Yaskawa INFORM job: ARIEL_TEST.JBI

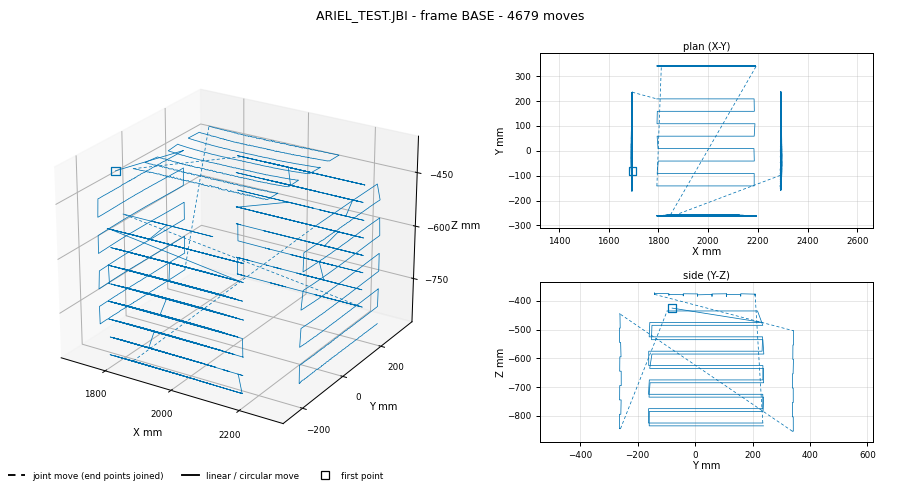
[picture p0: tool path of ARIEL_TEST.JBI in frame BASE, 4679 of 4679 moves have a stored position in this frame; points joined in program order, loops and branches not executed]
/JOB
//NAME ARIEL_TEST
//POS
///NPOS 4679,0,0,0,0,0
///TOOL 0
///POSTYPE BASE
///RECTAN
///RCONF 1,0,0,0,0,0,0,0,0,0,0,0,0,0,0,0,0,0,0,0,0,0,0,0
C00000=1696.132,-80.047,-425.128,-2.7960,72.8573,-92.9280
C00001=1694.988,235.674,-475.128,91.6331,81.5548,1.6157
C00002=1694.763,232.398,-475.128,113.1075,87.8917,23.0901
C00003=1694.793,228.055,-475.128,-70.6571,88.5964,-160.6630
C00004=1695.151,224.781,-475.128,-66.4401,88.6995,-156.4461
C00005=1695.130,221.009,-475.128,-43.9344,88.9803,-133.9346
C00006=1695.054,219.997,-475.128,-8.9266,88.7912,-98.9268
C00007=1695.058,217.094,-475.128,-159.0817,88.5678,110.9246
C00008=1694.887,215.803,-475.128,-11.6768,88.8428,-101.6770
C00009=1695.188,212.462,-475.128,-4.3716,86.4536,-94.3776
C00010=1695.133,208.131,-475.128,-42.6337,89.3986,-132.6340
C00011=1695.189,206.048,-475.128,-13.4931,89.5876,-103.4933
C00012=1695.116,201.470,-475.128,50.1911,88.5907,-39.8033
C00013=1694.965,197.460,-475.128,48.4607,89.2725,-41.5394
C00014=1695.140,191.185,-475.128,17.4924,89.6392,-72.5020
C00015=1694.918,187.331,-475.128,31.8851,88.8600,-58.1093
C00016=1695.110,184.389,-475.128,64.8530,89.3642,-25.1471
C00017=1694.969,179.240,-475.128,-12.1008,87.9146,-102.1068
C00018=1695.056,175.417,-475.128,38.8981,88.5907,-51.0906
C00019=1694.747,170.987,-475.128,47.6299,87.8172,-42.3473
C00020=1694.650,164.775,-475.128,16.4324,88.5105,-73.5620
C00021=1694.533,162.575,-475.128,42.0894,88.3901,-47.8992
C00022=1694.373,158.045,-475.128,56.9978,88.5563,-32.9909
C00023=1695.089,155.989,-475.128,-6.3483,88.3443,-96.3543
C00024=1695.185,152.477,-475.128,-65.8099,88.1495,-155.8216
C00025=1694.724,149.203,-475.128,6.0332,87.2614,-83.9612
C00026=1695.104,146.728,-475.128,19.4862,88.9230,-70.5139
C00027=1694.834,143.853,-475.128,47.7331,88.7053,-42.2556
C00028=1693.934,141.094,-475.128,115.7489,87.4906,25.7258
C00029=1693.799,137.257,-475.128,99.1904,86.6713,9.1730
C00030=1693.895,133.651,-475.128,38.0386,87.8287,-51.9386
C00031=1693.476,130.746,-475.128,21.7208,87.0265,-68.2507
C00032=1694.334,128.603,-475.128,25.3820,86.7859,-64.5838
C00033=1695.164,125.432,-475.128,143.9040,88.7110,53.8981
C00034=1694.863,121.656,-475.128,8.3823,87.0265,-81.6063
C00035=1693.391,117.740,-475.128,20.0649,87.7484,-69.9237
C00036=1694.429,115.474,-475.128,6.2051,87.3817,-83.7893
C00037=1693.264,112.358,-475.128,47.6242,88.3500,-42.3644
C00038=1694.551,109.480,-475.128,-7.0531,87.5078,-97.0590
C00039=1694.104,106.646,-475.128,8.1417,87.1984,-81.8470
C00040=1693.197,102.981,-475.128,-2.9507,87.4448,-92.9509
C00041=1694.004,100.489,-475.128,16.0313,86.9291,-73.9516
C00042=1694.629,96.503,-475.128,0.4354,86.7859,-89.5590
C00043=1693.339,94.279,-475.128,4.1539,86.6025,-85.8405
C00044=1693.243,89.591,-475.128,30.0688,88.3959,-59.9199
C00045=1694.046,86.533,-475.128,-0.4354,87.1010,-90.4356
C00046=1694.079,83.430,-475.128,-14.8969,86.6369,-104.9200
C00047=1694.640,81.259,-475.128,-7.5916,81.0620,-97.6835
C00048=1693.579,77.591,-475.128,-3.7013,86.7286,-93.7072
C00049=1694.579,74.118,-475.128,8.0615,86.6770,-81.9272
C00050=1694.602,71.620,-475.128,5.6550,86.3791,-84.3336
C00051=1693.230,67.936,-475.128,7.5745,86.6827,-82.4085
C00052=1692.692,63.461,-475.128,3.3689,87.3015,-86.6254
C00053=1693.515,60.204,-475.128,-3.5408,86.7515,-93.5410
C00054=1694.397,57.070,-475.128,-1.8678,86.3218,-91.8737
C00055=1695.083,51.313,-475.128,-46.0772,88.8542,-136.0832
C00056=1693.552,49.260,-475.128,3.4492,86.3275,-86.5452
C00057=1693.236,43.220,-475.128,-9.1501,86.3619,-99.1675
C00058=1692.438,40.123,-475.128,-10.2502,86.8604,-100.2676
C00059=1693.005,36.124,-475.128,-0.4583,86.2817,-90.4585
C00060=1694.308,31.082,-475.128,-2.0511,86.4937,-92.0571
C00061=1692.704,27.503,-475.128,2.7845,87.7828,-87.2099
C00062=1693.177,25.817,-475.128,10.8804,87.3073,-79.1082
C00063=1692.952,22.582,-475.128,5.8269,86.0525,-84.1617
C00064=1693.146,20.159,-475.128,3.7700,88.0636,-86.2244
C00065=1694.605,16.625,-475.128,-10.1413,85.7545,-100.1702
C00066=1693.774,12.699,-475.128,-8.9782,86.9578,-98.9899
C00067=1694.221,10.877,-475.128,9.3965,85.4566,-80.5693
C00068=1693.353,8.692,-475.128,-10.5882,87.4791,-100.5999
C00069=1695.395,6.553,-475.128,-14.2781,75.9627,-104.6965
C00070=1694.514,2.859,-475.128,-3.7757,86.2931,-93.7817
C00071=1694.492,-1.569,-475.128,-24.3277,87.2843,-114.3566
C00072=1692.776,-3.735,-475.128,-27.3186,87.2614,-117.3474
C00073=1694.690,-6.961,-475.128,-12.0607,85.7889,-102.0896
C00074=1694.113,-9.973,-475.128,-4.8816,87.4104,-94.8875
C00075=1695.315,-12.616,-475.128,5.5233,88.3386,-84.4711
C00076=1693.186,-16.477,-475.128,-14.8109,86.9692,-104.8283
C00077=1694.776,-17.860,-475.128,-8.1474,86.3963,-98.1591
C00078=1693.169,-22.210,-475.128,-23.4912,87.5364,-113.5086
C00079=1694.236,-24.585,-475.128,-9.7632,86.0238,-99.7863
C00080=1693.849,-28.361,-475.128,-19.7842,87.2041,-109.8073
C00081=1694.081,-32.852,-475.128,-27.7884,87.3932,-117.8173
C00082=1694.169,-36.280,-475.128,-40.8805,87.2156,-130.9151
C00083=1694.436,-38.893,-475.128,-11.4935,86.3332,-101.5166
C00084=1693.377,-42.844,-475.128,-15.4297,87.0208,-105.4528
C00085=1693.729,-46.013,-475.128,-5.6894,87.2843,-95.6954
C00086=1693.512,-48.882,-475.128,-21.3197,87.2729,-111.3371
C00087=1694.121,-53.479,-475.128,-2.0970,87.3703,-92.0972
C00088=1694.254,-55.606,-475.128,-8.6631,87.1239,-98.6747
C00089=1695.480,-60.498,-475.128,-7.5515,88.3615,-97.5517
C00090=1694.880,-63.263,-475.128,-10.0668,86.3447,-100.0899
C00091=1695.519,-67.371,-475.128,-4.2799,86.4650,-94.2916
C00092=1695.154,-69.634,-475.128,-16.6902,86.9062,-106.7133
C00093=1694.837,-73.212,-475.128,-14.3468,87.2099,-104.3642
C00094=1695.406,-77.363,-475.128,-22.5057,86.9921,-112.5346
C00095=1695.106,-81.047,-475.128,-14.6963,88.1438,-104.7023
C00096=1694.416,-84.097,-475.128,-20.3170,87.6281,-110.3344
C00097=1695.519,-87.829,-475.128,82.5403,88.9860,-7.4599
C00098=1694.707,-90.627,-475.128,-9.6600,86.9119,-99.6717
C00099=1695.330,-93.501,-475.128,-21.3369,87.6797,-111.3543
C00100=1695.363,-99.305,-475.128,-13.2009,87.5823,-103.2126
C00101=1694.622,-103.431,-475.128,-32.7502,88.3157,-122.7619
C00102=1695.475,-107.547,-475.128,2.7100,87.8401,-87.2901
C00103=1694.908,-111.406,-475.128,-12.5363,88.2355,-102.5422
C00104=1695.600,-115.157,-475.128,63.4035,89.7939,-26.5967
C00105=1694.895,-121.393,-475.128,-19.4691,88.3730,-109.4750
C00106=1695.267,-125.384,-475.128,-1.8907,88.4245,-91.8967
C00107=1694.736,-129.294,-475.128,-21.9041,89.0491,-111.9101
C00108=1694.843,-133.799,-475.128,-11.6940,88.3558,-101.6942
C00109=1695.271,-139.102,-475.128,-14.4328,88.7511,-104.4387
C00110=1695.095,-144.244,-475.128,-2.4751,88.2813,-92.4753
C00111=1694.850,-148.261,-475.128,-17.9851,88.4532,-107.9910
C00112=1695.327,-150.030,-475.128,46.9596,88.7855,-43.0348
C00113=1695.394,-153.452,-475.128,127.4143,87.1927,37.3854
C00114=1694.805,-157.684,-475.128,-67.2767,86.9635,-157.3055
C00115=1694.500,-159.876,-525.128,-78.9249,82.7121,-169.0110
C00116=1694.421,-156.702,-525.128,-95.0365,88.5391,174.9641
C00117=1694.689,-153.571,-525.128,-16.8220,89.4845,-106.8222
C00118=1694.622,-150.053,-525.128,-18.9878,88.8657,-108.9937
C00119=1694.362,-147.366,-525.128,-40.2216,88.8657,-130.2218
C00120=1694.470,-144.581,-525.128,-53.1189,88.8428,-143.1248
C00121=1694.487,-142.921,-525.128,-69.2419,88.9115,-159.2478
C00122=1694.727,-138.966,-525.128,-58.3614,89.2381,-148.3674
C00123=1694.454,-135.239,-525.128,-40.0268,88.5735,-130.0327
C00124=1694.239,-130.327,-525.128,-74.8282,88.7397,-164.8342
C00125=1694.291,-126.172,-525.128,-35.7353,88.3271,-125.7470
C00126=1693.961,-120.293,-525.128,-44.4557,88.1610,-134.4674
C00127=1694.229,-117.327,-525.128,-39.6773,88.3787,-129.6889
C00128=1693.955,-112.124,-525.128,-39.0126,88.5506,-129.0186
C00129=1694.120,-109.056,-525.128,-37.0875,88.5448,-127.0992
C00130=1693.350,-104.310,-525.128,-49.8072,87.8401,-139.8246
C00131=1693.551,-100.440,-525.128,-37.3396,87.8000,-127.3570
C00132=1693.489,-95.539,-525.128,-61.2778,87.2328,-151.3066
C00133=1693.865,-92.922,-525.128,-39.5627,87.4390,-129.5915
C00134=1693.249,-88.499,-525.128,-41.9175,88.7740,-131.9235
C00135=1693.006,-86.270,-525.128,-63.5410,88.3730,-153.5469
C00136=1693.393,-79.718,-525.128,-36.8870,87.8573,-126.9044
C00137=1693.031,-76.883,-525.128,-29.2265,87.6510,-119.2497
C00138=1693.235,-73.650,-525.128,-33.6670,87.9432,-123.6843
C00139=1692.490,-67.602,-525.128,-23.0443,87.4963,-113.0617
C00140=1693.098,-63.993,-525.128,-33.1627,87.5021,-123.1916
C00141=1692.056,-60.055,-525.128,-46.8564,88.6537,-136.8624
C00142=1692.699,-57.465,-525.128,-34.4118,88.1724,-124.4235
C00143=1692.339,-53.601,-525.128,-27.2154,88.0349,-117.2271
C00144=1692.501,-49.582,-525.128,-18.1570,88.0922,-108.1687
C00145=1691.991,-47.866,-525.128,-46.9997,88.2927,-137.0171
C00146=1692.189,-44.341,-525.128,-17.3835,87.7599,-107.3952
C00147=1691.755,-40.515,-525.128,-28.3900,88.4646,-118.4017
C00148=1692.760,-37.856,-525.128,-26.7571,86.3218,-116.8031
C00149=1692.377,-34.007,-525.128,-22.9297,88.8313,-112.9299
C00150=1692.333,-29.550,-525.128,-22.8438,88.3558,-112.8497
C00151=1691.906,-26.667,-525.128,-25.7831,88.2125,-115.7947
C00152=1692.601,-23.052,-525.128,-46.5069,87.6510,-136.5301
C00153=1691.715,-19.895,-525.128,-46.5241,88.3787,-136.5358
C00154=1691.346,-17.017,-525.128,-23.3709,88.2698,-113.3826
C00155=1691.553,-15.002,-525.128,-34.4233,88.3500,-124.4349
C00156=1691.985,-9.968,-525.128,-10.4163,88.0750,-100.4223
C00157=1691.467,-6.304,-525.128,-5.8097,88.0235,-95.8157
C00158=1691.911,-3.077,-525.128,-20.7468,88.7167,-110.7527
C00159=1691.862,0.698,-525.128,-8.0729,88.0521,-98.0789
C00160=1691.612,3.808,-525.128,-39.1272,89.0491,-129.1274
C00161=1692.269,7.928,-525.128,-24.4309,87.2041,-114.4540
C00162=1691.326,9.877,-525.128,-26.0180,88.9287,-116.0239
C00163=1691.066,12.948,-525.128,-66.2682,87.8287,-156.2799
C00164=1691.291,15.880,-525.128,-9.7345,87.5193,-99.7462
C00165=1691.603,21.223,-525.128,-14.0145,88.6594,-104.0204
C00166=1691.244,23.875,-525.128,20.1165,88.7282,-69.8779
C00167=1691.672,27.568,-525.128,-40.1414,88.2584,-130.1530
C00168=1691.918,29.995,-525.128,-5.0305,87.2958,-95.0365
C00169=1691.532,34.742,-525.128,62.2805,89.2725,-27.7139
C00170=1691.777,36.968,-525.128,1.6386,87.6338,-88.3615
C00171=1692.094,41.761,-525.128,7.4656,88.8428,-82.5288
C00172=1692.187,44.735,-525.128,16.2433,87.9375,-73.7453
C00173=1691.171,47.416,-525.128,33.8675,88.9688,-56.1326
C00174=1691.446,51.083,-525.128,10.5825,88.5047,-79.4176
C00175=1691.301,52.729,-525.128,50.8156,89.1636,-39.1788
C00176=1691.411,56.907,-525.128,101.2760,88.8084,11.2700
C00177=1691.256,60.771,-525.128,20.4202,88.4876,-69.5742
C00178=1691.909,62.038,-525.128,2.8074,88.3901,-87.1927
C00179=1692.124,67.281,-525.128,17.0626,88.3500,-72.9317
C00180=1692.099,70.838,-525.128,26.3732,88.4417,-63.6155
C00181=1692.157,72.684,-525.128,18.6497,88.3787,-71.3389
C00182=1691.565,76.598,-525.128,3.0366,88.4646,-86.9635
C00183=1691.909,80.224,-525.128,105.0174,89.1235,15.0172
C00184=1692.286,84.108,-525.128,18.7185,88.2985,-71.2759
C00185=1691.948,86.578,-525.128,38.0386,88.4303,-51.9500
C00186=1691.934,90.287,-525.128,18.0309,88.6079,-71.9634
C00187=1692.085,93.239,-525.128,42.8687,88.0406,-47.1143
C00188=1692.449,96.809,-525.128,-8.6000,87.5651,-98.6117
C00189=1691.972,100.726,-525.128,51.9328,88.3271,-38.0558
C00190=1692.777,102.244,-525.128,51.5031,87.0036,-38.4569
C00191=1692.585,107.563,-525.128,43.8312,88.0521,-46.1517
C00192=1692.245,109.667,-525.128,90.3153,88.5620,0.3151
C00193=1692.710,113.138,-525.128,77.6587,88.0177,-12.3300
C00194=1692.487,115.926,-525.128,54.4367,88.4417,-35.5520
C00195=1692.585,119.868,-525.128,70.5425,88.5506,-19.4519
C00196=1692.703,124.136,-525.128,68.0387,87.8573,-21.9500
C00197=1693.348,127.989,-525.128,14.1234,89.0089,-75.8710
C00198=1693.014,131.500,-525.128,52.6891,87.9604,-37.2938
C00199=1693.004,135.286,-525.128,69.1903,88.0235,-20.7983
C00200=1693.062,138.337,-525.128,70.2961,88.6709,-19.6982
C00201=1693.695,142.853,-525.128,36.3083,87.1640,-53.6574
C00202=1693.927,146.038,-525.128,25.0325,87.9261,-64.9562
C00203=1693.303,150.565,-525.128,86.1900,88.5907,-3.8101
C00204=1693.469,156.957,-525.128,171.4862,89.6621,81.4860
C00205=1693.614,160.194,-525.128,68.4799,88.0578,-21.5088
C00206=1693.876,164.625,-525.128,83.0502,88.7454,-6.9499
C00207=1694.292,168.627,-525.128,69.0127,88.8313,-20.9874
C00208=1693.978,172.496,-525.128,66.4229,88.3901,-23.5657
C00209=1694.116,176.139,-525.128,93.7931,88.9918,3.7929
C00210=1694.081,181.483,-525.128,58.4187,88.5506,-31.5699
C00211=1694.426,184.221,-525.128,61.7419,88.6480,-28.2525
C00212=1694.402,190.301,-525.128,32.2174,89.0089,-57.7770
C00213=1694.649,195.955,-525.128,59.7652,88.7225,-30.2292
C00214=1694.804,197.877,-525.128,52.6376,89.0261,-37.3568
C00215=1694.710,202.217,-525.128,65.4546,89.3241,-24.5455
C00216=1694.828,206.371,-525.128,47.6127,89.0147,-42.3816
C00217=1694.680,209.763,-525.128,130.3364,88.5792,40.3247
C00218=1694.784,212.216,-525.128,55.0211,88.9173,-34.9790
C00219=1694.849,214.324,-525.128,1.7475,87.8802,-88.2526
C00220=1694.724,215.988,-525.128,31.4038,88.4818,-58.5849
C00221=1694.889,219.187,-525.128,4.8987,88.7454,-85.1014
C00222=1694.788,221.768,-525.128,-122.8306,84.2477,147.3017
C00223=1694.756,224.941,-525.128,-136.6045,88.2698,133.4074
C00224=1694.729,227.663,-525.128,7.0817,89.8225,-82.9184
C00225=1694.687,230.259,-525.128,50.5119,89.1350,-39.4882
C00226=1694.723,234.923,-525.128,92.3550,83.3539,2.3376
C00227=1694.806,233.203,-575.128,103.6537,82.6205,13.5447
C00228=1694.742,231.059,-575.128,75.1204,86.9520,-14.8625
C00229=1694.693,226.262,-575.128,-78.3691,89.0089,-168.3693
C00230=1694.887,224.564,-575.128,-9.8663,89.8627,-99.8665
C00231=1694.695,221.286,-575.128,-22.9068,89.4788,-112.9070
C00232=1694.713,219.344,-575.128,73.4646,89.3871,-16.5355
C00233=1694.584,216.524,-575.128,139.2974,89.7251,49.2972
C00234=1694.630,213.463,-575.128,27.1295,88.9688,-62.8706
C00235=1694.668,210.962,-575.128,162.0611,88.7282,72.0551
C00236=1694.607,208.721,-575.128,108.3577,89.0491,18.3575
C00237=1694.629,206.423,-575.128,24.9351,89.0949,-65.0650
C00238=1694.628,202.253,-575.128,69.9524,89.2209,-20.0420
C00239=1694.515,199.405,-575.128,104.0892,89.1121,14.0833
C00240=1694.346,194.510,-575.128,53.2392,88.7912,-36.7552
C00241=1694.248,188.122,-575.128,78.4379,88.5277,-11.5565
C00242=1694.228,183.278,-575.128,96.9043,88.2240,6.9041
C00243=1693.970,179.423,-575.128,78.9535,88.2183,-11.0408
C00244=1693.868,172.668,-575.128,53.3538,88.5792,-36.6406
C00245=1693.812,169.950,-575.128,112.5231,88.3672,22.5172
C00246=1693.709,166.789,-575.128,79.9562,89.1063,-10.0382
C00247=1693.646,162.728,-575.128,71.4707,88.2125,-18.5179
C00248=1693.661,159.420,-575.128,85.0555,88.2068,-4.9388
C00249=1693.425,155.227,-575.128,91.6961,88.0349,1.6959
C00250=1693.320,151.517,-575.128,78.8619,88.6480,-11.1325
C00251=1693.201,147.367,-575.128,74.5876,88.3901,-15.4068
C00252=1692.996,142.122,-575.128,106.0430,87.4963,16.0313
C00253=1692.897,140.572,-575.128,57.8744,88.1094,-32.1142
C00254=1692.852,136.432,-575.128,102.2328,86.9979,12.2154
C00255=1692.607,133.096,-575.128,108.3119,88.1667,18.3002
C00256=1692.506,127.929,-575.128,84.0070,88.0979,-5.9874
C00257=1692.637,126.345,-575.128,103.8142,88.4876,13.8082
C00258=1692.460,120.405,-575.128,121.4269,87.8917,31.4095
C00259=1692.265,116.228,-575.128,86.4650,88.6365,-3.5351
C00260=1692.250,112.447,-575.128,102.2786,88.5105,12.2727
C00261=1692.136,109.594,-575.128,72.0551,88.4131,-17.9335
C00262=1691.893,104.059,-575.128,56.6941,88.4761,-33.2945
C00263=1691.813,101.461,-575.128,106.7821,88.6365,16.7819
C00264=1691.820,97.498,-575.128,48.3003,88.7167,-41.6941
C00265=1691.695,93.109,-575.128,97.0074,88.6423,7.0072
C00266=1691.744,90.048,-575.128,96.6866,88.6709,6.6864
C00267=1691.683,85.860,-575.128,134.9888,88.6021,44.9829
C00268=1691.585,83.286,-575.128,85.6400,89.3642,-4.3602
C00269=1691.337,79.352,-575.128,57.0436,88.7282,-32.9508
C00270=1691.369,74.414,-575.128,75.4241,89.2553,-14.5760
C00271=1691.218,72.542,-575.128,119.8627,89.6105,29.8625
C00272=1691.295,67.757,-575.128,66.8527,89.1063,-23.1474
C00273=1691.304,64.282,-575.128,163.5794,87.8287,73.5677
C00274=1691.097,62.191,-575.128,56.9921,89.1522,-33.0023
C00275=1690.987,56.823,-575.128,-140.2256,89.2840,129.7749
C00276=1691.165,55.524,-575.128,34.3831,88.3672,-55.6055
C00277=1691.027,51.901,-575.128,118.2298,89.7251,28.2296
C00278=1690.928,47.456,-575.128,56.2415,88.6537,-33.7472
C00279=1690.984,45.810,-575.128,-8.4625,88.2985,-98.4685
C00280=1691.087,41.819,-575.128,-52.0302,89.1465,-142.0362
C00281=1691.043,39.213,-575.128,142.3055,89.5131,52.3053
C00282=1691.026,35.327,-575.128,-28.4874,89.5647,-118.4876
C00283=1690.873,32.032,-575.128,45.8480,89.1808,-44.1521
C00284=1690.821,30.213,-575.128,33.9133,88.1610,-56.0696
C00285=1690.929,26.425,-575.128,-12.6623,88.6136,-102.6683
C00286=1690.815,23.772,-575.128,-111.9043,89.3355,158.0962
C00287=1690.808,19.852,-575.128,57.7598,89.6105,-32.2403
C00288=1690.950,16.612,-575.128,-115.5254,89.8569,154.4751
C00289=1690.737,11.905,-575.128,-109.0395,88.8944,160.9667
C00290=1690.920,8.527,-575.128,-84.2706,89.0261,-174.2708
C00291=1690.739,5.954,-575.128,167.0458,89.8856,77.0456
C00292=1690.841,2.739,-575.128,-19.8128,89.6277,-109.8130
C00293=1690.672,-1.372,-575.128,31.7705,89.5819,-58.2297
C00294=1690.806,-3.662,-575.128,-41.4706,88.4646,-131.4766
C00295=1691.056,-8.688,-575.128,-28.0290,89.0491,-118.0293
C00296=1690.987,-12.668,-575.128,6.5145,88.8141,-83.4856
C00297=1690.795,-20.036,-575.128,-41.3446,89.4329,-131.3448
C00298=1690.997,-24.547,-575.128,-76.8909,89.0491,-166.8968
C00299=1690.918,-30.269,-575.128,-25.9664,89.1350,-115.9723
C00300=1691.294,-35.152,-575.128,-25.2960,88.2240,-115.3020
C00301=1691.022,-39.070,-575.128,-46.2949,89.0376,-136.3009
C00302=1691.086,-41.699,-575.128,-46.7991,88.7626,-136.8051
C00303=1691.265,-47.309,-575.128,-46.3465,88.8485,-136.3524
C00304=1691.355,-50.600,-575.128,-19.8644,88.9918,-109.8646
C00305=1691.892,-55.259,-575.128,-41.7514,88.0750,-131.7631
C00306=1691.475,-59.480,-575.128,-78.1113,88.1782,-168.1172
C00307=1691.274,-63.897,-575.128,-78.4723,88.2125,-168.4782
C00308=1691.851,-66.924,-575.128,-38.8236,87.9662,-128.8410
C00309=1691.543,-71.041,-575.128,-128.1935,87.8000,141.8299
C00310=1691.724,-73.351,-575.128,-3.1111,88.0292,-93.1113
C00311=1692.211,-78.850,-575.128,-89.1235,88.8772,-179.1237
C00312=1692.125,-79.622,-575.128,-76.7820,88.8371,-166.7880
C00313=1692.001,-84.001,-575.128,-76.4382,88.6480,-166.4385
C00314=1692.577,-87.866,-575.128,-56.2587,88.8256,-146.2589
C00315=1692.045,-91.980,-575.128,-95.6209,88.5792,174.3797
C00316=1692.173,-94.043,-575.128,-85.5082,87.7771,-175.5084
C00317=1692.553,-100.118,-575.128,-73.2984,88.1094,-163.3044
C00318=1692.848,-103.049,-575.128,-65.8099,88.1438,-155.8216
C00319=1693.065,-107.930,-575.128,-76.1518,87.5135,-166.1634
C00320=1692.948,-112.113,-575.128,-59.5646,88.7339,-149.5706
C00321=1693.011,-116.306,-575.128,-82.8153,88.0005,-172.8155
C00322=1693.309,-121.879,-575.128,-72.7656,87.0552,-162.7887
C00323=1693.330,-125.985,-575.128,-81.2282,87.4104,-171.2341
C00324=1693.636,-128.998,-575.128,-81.9501,88.0521,-171.9503
C00325=1693.762,-132.765,-575.128,-79.5609,88.3042,-169.5668
C00326=1693.867,-137.386,-575.128,-126.5606,88.6480,143.4457
C00327=1694.041,-140.149,-575.128,-69.7919,88.0693,-159.8036
C00328=1694.038,-142.787,-575.128,-94.8130,88.0578,175.1875
C00329=1694.000,-144.618,-575.128,-71.5337,87.9662,-161.5454
C00330=1694.203,-147.692,-575.128,-95.3344,88.5735,174.6661
C00331=1694.311,-152.225,-575.128,-102.1755,89.2553,167.8250
C00332=1694.376,-154.259,-575.128,31.0600,89.7194,-58.9401
C00333=1694.414,-156.252,-575.128,-114.2477,87.3416,155.7757
C00334=1694.517,-158.357,-575.128,-103.1839,88.8886,166.8223
C00335=1694.945,-161.433,-575.128,-94.7385,78.2603,175.3594
C00336=1694.553,-161.479,-625.128,-68.8065,79.0509,-159.1562
C00337=1694.756,-158.430,-625.128,-76.2205,83.7607,-166.3010
C00338=1694.559,-156.743,-625.128,-104.3871,86.4134,165.6363
C00339=1694.303,-153.567,-625.128,-61.5643,87.5594,-151.5874
C00340=1694.320,-150.343,-625.128,-84.2992,87.4505,-174.2994
C00341=1693.989,-147.719,-625.128,-78.0139,86.9921,-168.0313
C00342=1693.810,-142.914,-625.128,-75.4814,87.1010,-165.4988
C00343=1693.818,-139.261,-625.128,-95.1109,87.3703,174.8953
C00344=1693.699,-134.943,-625.128,-92.1201,88.0235,177.8804
C00345=1693.573,-130.480,-625.128,-96.1194,87.6453,173.8869
C00346=1693.153,-126.406,-625.128,-86.9463,87.1239,-176.9522
C00347=1693.106,-121.856,-625.128,-78.7186,87.0953,-168.7303
C00348=1692.960,-118.089,-625.128,-84.1331,87.9261,-174.1390
C00349=1692.713,-112.713,-625.128,-82.2480,87.9719,-172.2540
C00350=1692.412,-110.341,-625.128,-74.7022,88.2469,-164.7081
C00351=1692.432,-106.464,-625.128,-76.3580,88.2125,-166.3640
C00352=1692.347,-102.865,-625.128,-97.5747,88.0464,172.4316
C00353=1692.024,-98.807,-625.128,-67.6605,87.7255,-157.6779
C00354=1692.063,-93.005,-625.128,-73.8599,88.8600,-163.8602
C00355=1692.032,-88.429,-625.128,-83.3539,87.9547,-173.3541
C00356=1691.922,-85.154,-625.128,-81.5777,87.8974,-171.5836
C00357=1691.639,-80.293,-625.128,-118.3329,88.1037,151.6791
C00358=1691.561,-76.884,-625.128,-63.2258,88.4990,-153.2375
C00359=1691.419,-71.985,-625.128,-22.7693,86.4593,-112.8096
C00360=1691.352,-67.828,-625.128,-54.3163,88.7969,-144.3223
C00361=1691.103,-64.509,-625.128,-48.2315,88.3730,-138.2375
C00362=1691.180,-61.617,-625.128,-24.0012,88.9975,-114.0014
C00363=1691.089,-57.626,-625.128,-73.8198,88.9287,-163.8200
C00364=1691.159,-54.104,-625.128,151.6561,89.9257,61.6559
C00365=1691.154,-50.557,-625.128,-38.6746,89.0204,-128.6748
C00366=1691.026,-48.692,-625.128,-45.7220,88.6652,-135.7279
C00367=1690.951,-44.611,-625.128,-74.4214,89.0147,-164.4216
C00368=1690.795,-42.130,-625.128,-39.3335,88.9574,-129.3337
C00369=1690.759,-37.278,-625.128,-49.5322,89.4673,-139.5324
C00370=1690.847,-34.944,-625.128,-94.3718,89.3699,175.6287
C00371=1690.742,-31.427,-625.128,-121.1290,89.4559,148.8716
C00372=1690.778,-28.339,-625.128,-12.2784,89.0204,-102.2786
C00373=1690.609,-25.061,-625.128,40.0497,89.7481,-49.9447
C00374=1690.613,-21.692,-625.128,124.7329,89.0433,34.7269
C00375=1690.768,-19.120,-625.128,-153.7188,88.7568,116.2875
C00376=1690.638,-13.464,-625.128,-174.7463,89.0319,95.2542
C00377=1690.663,-8.718,-625.128,151.9083,89.5361,61.9080
C00378=1690.737,-6.140,-625.128,-21.6635,89.3527,-111.6637
C00379=1690.630,-4.212,-625.128,-49.5665,89.3241,-139.5667
C00380=1690.744,-0.158,-625.128,-167.3896,88.9345,102.6110
C00381=1690.633,2.934,-625.128,54.8893,88.9001,-35.1051
C00382=1690.812,6.829,-625.128,19.4232,89.4444,-70.5769
C00383=1690.813,11.135,-625.128,109.5896,89.4845,19.5894
C00384=1690.874,15.819,-625.128,-149.2096,89.4501,120.7966
C00385=1691.095,20.063,-625.128,104.0090,88.0177,14.0030
C00386=1690.840,22.530,-625.128,95.6553,89.3298,5.6550
C00387=1690.961,26.623,-625.128,68.8695,88.7912,-21.1249
C00388=1690.939,30.121,-625.128,56.7514,89.3928,-33.2487
C00389=1690.878,33.744,-625.128,40.2159,88.9230,-49.7843
C00390=1690.938,36.801,-625.128,175.4052,89.4960,85.4050
C00391=1690.897,40.528,-625.128,-120.2122,89.8970,149.7826
C00392=1691.261,42.787,-625.128,84.9581,88.8829,-5.0420
C00393=1691.064,46.432,-625.128,75.6533,89.3126,-14.3411
C00394=1691.059,50.483,-625.128,168.7188,88.8829,78.7186
C00395=1691.194,54.245,-625.128,115.2160,88.8141,25.2158
C00396=1691.318,58.791,-625.128,99.2477,89.1407,9.2475
C00397=1691.361,61.495,-625.128,88.2813,88.3443,-1.7188
C00398=1691.203,66.319,-625.128,136.7077,88.4818,46.6960
C00399=1691.260,69.455,-625.128,-114.0644,89.4730,155.9361
C00400=1691.776,71.904,-625.128,122.2806,89.2897,32.2747
C00401=1691.544,76.312,-625.128,138.5870,88.0578,48.5753
C00402=1691.652,79.136,-625.128,143.6691,88.1953,53.6574
C00403=1691.489,81.695,-625.128,24.7059,88.7798,-65.2885
C00404=1691.825,84.982,-625.128,86.7286,88.4646,-3.2715
C00405=1691.761,87.171,-625.128,83.0273,88.5506,-6.9728
C00406=1691.764,91.864,-625.128,125.2485,88.5506,35.2369
C00407=1691.811,95.976,-625.128,111.2855,87.9490,21.2739
C00408=1692.051,97.972,-625.128,81.9157,88.9173,-8.0787
C00409=1692.046,101.259,-625.128,54.7403,87.8057,-35.2426
C00410=1692.323,105.961,-625.128,131.6026,88.5735,41.5967
C00411=1692.101,108.639,-625.128,117.5823,88.4704,27.5764
C00412=1692.376,112.436,-625.128,114.3910,87.3932,24.3736
C00413=1692.334,115.215,-625.128,93.3520,87.9089,3.3518
C00414=1692.524,118.458,-625.128,89.3928,88.9803,-0.6073
C00415=1692.672,121.812,-625.128,85.1930,88.7282,-4.8071
C00416=1692.830,126.268,-625.128,118.7225,88.5448,28.7166
C00417=1692.865,130.574,-625.128,142.6091,88.8542,52.6032
C00418=1693.032,134.375,-625.128,98.4226,88.2813,8.4167
C00419=1692.945,136.693,-625.128,128.8295,87.8344,38.8064
C00420=1693.180,141.376,-625.128,45.4813,88.2526,-44.5016
C00421=1692.988,143.518,-625.128,17.8762,88.3443,-72.1124
C00422=1693.249,148.889,-625.128,46.5814,88.3443,-43.4072
C00423=1693.385,151.667,-625.128,24.1100,88.5907,-65.8844
C00424=1693.535,156.208,-625.128,77.9910,88.3042,-12.0034
C00425=1693.629,160.429,-625.128,100.0785,88.6365,10.0725
C00426=1693.584,162.586,-625.128,79.7156,88.6881,-10.2788
C00427=1693.916,167.276,-625.128,-126.3773,88.8886,143.6290
C00428=1693.851,170.854,-625.128,82.5345,88.4303,-7.4599
C00429=1694.063,174.582,-625.128,120.3268,88.4990,30.3151
C00430=1693.968,177.425,-625.128,66.0333,89.0892,-23.9668
C00431=1694.060,181.015,-625.128,61.6731,88.9574,-28.3213
C00432=1694.049,183.667,-625.128,81.9043,88.6881,-8.0901
C00433=1694.155,186.522,-625.128,58.6995,87.9375,-31.2834
C00434=1694.273,190.850,-625.128,64.3317,89.5074,-25.6685
C00435=1694.261,194.576,-625.128,80.5578,88.8256,-9.4366
C00436=1694.375,196.487,-625.128,75.6991,88.7339,-14.3010
C00437=1694.430,199.264,-625.128,114.8436,88.5735,24.8377
C00438=1694.342,202.564,-625.128,41.4477,89.6908,-48.5524
C00439=1694.471,206.831,-625.128,54.7346,89.1751,-35.2598
C00440=1694.648,209.887,-625.128,-95.4948,89.7767,174.5057
C00441=1694.667,213.074,-625.128,94.5609,88.8199,4.5607
C00442=1694.646,215.930,-625.128,158.3426,89.0777,68.3424
C00443=1694.487,218.634,-625.128,130.1015,89.4215,40.0955
C00444=1694.698,222.258,-625.128,139.6928,88.4131,49.6869
C00445=1694.679,225.429,-625.128,173.0389,89.0319,83.0330
C00446=1694.702,227.521,-625.128,-120.7393,88.2068,149.2726
C00447=1694.633,230.367,-625.128,84.6831,89.2610,-5.3170
C00448=1694.651,232.143,-625.128,89.3241,87.5193,-0.6760
C00449=1694.803,234.775,-625.128,94.5036,78.2030,4.4117
C00450=1695.065,235.983,-625.128,95.1511,74.3298,4.9560
C00451=1695.245,235.879,-675.128,93.5640,73.4818,3.4205
C00452=1694.638,231.558,-675.128,126.8929,88.8600,36.8870
C00453=1694.621,230.657,-675.128,145.2390,89.0147,55.2388
C00454=1694.786,227.972,-675.128,116.4021,89.2381,26.3961
C00455=1694.835,225.201,-675.128,-99.4712,89.9257,170.5294
C00456=1694.776,222.095,-675.128,108.3119,88.8944,18.3060
C00457=1694.564,216.891,-675.128,75.4470,88.3844,-14.5473
C00458=1694.567,212.845,-675.128,70.2388,89.3814,-19.7613
C00459=1694.574,210.852,-675.128,73.3385,89.1579,-16.6616
C00460=1694.586,206.438,-675.128,119.4387,88.4474,29.4271
C00461=1694.540,204.609,-675.128,117.6053,88.9402,27.6051
C00462=1694.307,199.817,-675.128,93.6556,88.3214,3.6554
C00463=1694.179,195.707,-675.128,89.2439,89.0319,-0.7563
C00464=1694.211,192.151,-675.128,67.3340,89.3584,-22.6662
C00465=1694.109,188.180,-675.128,92.7847,88.4245,2.7845
C00466=1694.138,183.661,-675.128,82.6147,89.5991,-7.3854
C00467=1694.048,180.823,-675.128,73.1495,88.8542,-16.8449
C00468=1693.896,177.478,-675.128,87.5536,88.3787,-2.4465
C00469=1694.085,174.820,-675.128,132.1469,88.6251,42.1410
C00470=1693.776,169.386,-675.128,98.5086,88.4933,8.5026
C00471=1693.704,165.885,-675.128,106.6045,88.5850,16.5985
C00472=1693.611,162.289,-675.128,116.2989,89.0261,26.2930
C00473=1693.880,157.966,-675.128,134.8398,89.3355,44.8396
C00474=1693.699,154.392,-675.128,106.7649,89.3355,16.7647
C00475=1693.583,150.822,-675.128,43.8026,89.6220,-46.1975
C00476=1693.439,147.709,-675.128,114.7978,89.0147,24.7976
C00477=1693.225,145.601,-675.128,149.6336,88.4360,59.6277
C00478=1693.427,142.311,-675.128,78.3462,88.4016,-11.6539
C00479=1693.079,137.686,-675.128,110.7928,88.6881,20.7869
C00480=1692.987,136.923,-675.128,71.9806,89.6163,-18.0137
C00481=1693.339,131.791,-675.128,114.4254,88.3730,24.4194
C00482=1693.013,129.588,-675.128,141.8471,89.4387,51.8469
C00483=1692.767,125.654,-675.128,104.6049,88.7225,14.5989
C00484=1692.813,122.006,-675.128,102.1010,87.8573,12.0894
C00485=1692.812,119.181,-675.128,110.9933,89.1006,20.9874
C00486=1692.816,114.880,-675.128,134.2841,88.4704,44.2724
C00487=1692.599,111.705,-675.128,145.6458,89.4788,55.6456
C00488=1692.551,105.915,-675.128,138.8563,88.9173,48.8503
C00489=1692.353,103.666,-675.128,141.6179,88.6423,51.6063
C00490=1692.606,99.889,-675.128,136.3868,89.1579,46.3809
C00491=1692.461,95.053,-675.128,117.8402,89.1579,27.8400
C00492=1692.235,91.643,-675.128,101.1327,87.8172,11.1211
C00493=1692.499,87.954,-675.128,153.8219,87.6396,63.8045
C00494=1692.535,86.109,-675.128,80.0651,89.0089,-9.9350
C00495=1692.496,81.933,-675.128,179.9144,88.1037,89.9142
C00496=1691.996,77.963,-675.128,105.4586,88.8084,15.4584
C00497=1692.115,72.851,-675.128,93.9249,89.2152,3.9247
C00498=1692.245,70.999,-675.128,151.4040,87.6338,61.3866
C00499=1691.752,66.406,-675.128,102.7657,88.6480,12.7655
C00500=1692.183,63.371,-675.128,124.0682,88.5334,34.0623
C00501=1691.637,59.884,-675.128,62.0226,88.7454,-27.9718
C00502=1691.839,57.285,-675.128,133.7913,88.1037,43.7797
C00503=1691.528,53.894,-675.128,103.4704,89.0147,13.4702
C00504=1691.820,47.982,-675.128,110.6037,89.2209,20.6035
C00505=1691.923,45.596,-675.128,135.2237,87.8802,45.2063
C00506=1691.279,41.081,-675.128,129.1790,88.2355,39.1673
C00507=1691.624,35.574,-675.128,142.6951,89.0032,52.6891
C00508=1691.600,33.164,-675.128,136.7363,88.7798,46.7247
C00509=1690.980,26.763,-675.128,-18.5581,89.4272,-108.5583
C00510=1690.949,21.099,-675.128,107.5728,88.8256,17.5668
C00511=1691.143,16.194,-675.128,116.1671,89.0662,26.1669
C00512=1691.424,11.751,-675.128,133.7569,89.2496,43.7567
C00513=1691.094,7.273,-675.128,110.4834,88.2183,20.4717
C00514=1690.870,3.199,-675.128,150.4186,89.6564,60.4183
C00515=1690.954,-1.233,-675.128,141.7096,89.0433,51.7094
C00516=1690.851,-6.282,-675.128,113.3310,88.9688,23.3251
C00517=1691.009,-8.317,-675.128,107.9051,89.3814,17.9049
C00518=1690.981,-12.509,-675.128,140.8788,88.8313,50.8729
C00519=1690.792,-14.250,-675.128,121.7535,88.5448,31.7475
C00520=1690.997,-19.700,-675.128,130.1416,88.4073,40.1299
C00521=1690.764,-22.287,-675.128,-165.6249,89.1980,104.3757
C00522=1690.559,-24.595,-675.128,81.8584,89.4157,-8.1360
C00523=1690.630,-27.426,-675.128,-4.1081,89.7194,-94.1083
C00524=1690.758,-32.489,-675.128,-74.5819,89.8225,-164.5821
C00525=1690.754,-34.883,-675.128,175.6860,89.3298,85.6858
C00526=1690.749,-39.937,-675.128,-48.4321,89.7996,-138.4323
C00527=1690.725,-44.414,-675.128,-132.7944,89.4157,137.2062
C00528=1690.788,-47.195,-675.128,-58.6250,89.3069,-148.6252
C00529=1690.761,-51.141,-675.128,-113.9441,89.0949,156.0565
C00530=1690.857,-54.909,-675.128,-31.4611,89.4845,-121.4613
C00531=1690.932,-56.457,-675.128,-104.0147,89.2381,165.9916
C00532=1690.952,-62.657,-675.128,-60.4699,89.6163,-150.4701
C00533=1690.945,-67.080,-675.128,-115.8176,89.2897,154.1829
C00534=1690.993,-68.922,-675.128,-120.3211,88.8657,149.6852
C00535=1691.168,-74.266,-675.128,-71.3618,89.3871,-161.3621
C00536=1691.235,-77.564,-675.128,18.1684,89.1235,-71.8317
C00537=1691.168,-79.420,-675.128,-70.3764,89.3470,-160.3766
C00538=1691.279,-83.136,-675.128,-6.2223,89.2439,-96.2225
C00539=1691.188,-86.832,-675.128,-86.9749,89.1121,-176.9752
C00540=1691.324,-92.414,-675.128,-80.7755,88.8199,-170.7758
C00541=1691.540,-98.964,-675.128,-86.8604,88.0922,-176.8606
C00542=1691.811,-105.062,-675.128,-83.1934,87.9891,-173.1994
C00543=1692.210,-112.360,-675.128,-63.3232,87.8000,-153.3406
C00544=1692.209,-115.189,-675.128,-93.1171,88.2412,176.8835
C00545=1692.266,-119.780,-675.128,-77.7962,87.0609,-167.8136
C00546=1692.437,-123.193,-675.128,-84.9123,87.4390,-174.9182
C00547=1692.778,-128.012,-675.128,-71.0467,87.3416,-161.0641
C00548=1692.792,-133.918,-675.128,-85.9264,87.5708,-175.9266
C00549=1693.046,-136.595,-675.128,-101.6083,86.9635,168.4094
C00550=1693.198,-140.397,-675.128,-75.1147,86.9463,-165.1321
C00551=1693.224,-144.578,-675.128,-64.2285,88.0979,-154.2459
C00552=1693.395,-149.262,-675.128,-70.4680,87.2328,-160.4912
C00553=1693.731,-154.414,-675.128,-70.3706,88.4417,-160.3766
C00554=1694.180,-157.429,-675.128,-79.7213,85.9551,-169.7444
C00555=1694.113,-159.350,-675.128,-80.8328,84.3279,-170.8789
C00556=1693.613,-162.296,-725.128,-77.2920,71.8660,-167.9052
C00557=1693.452,-158.027,-725.128,-75.1262,87.1067,-165.1436
C00558=1693.478,-154.036,-725.128,-82.0475,88.6938,-172.0477
C00559=1693.526,-153.060,-725.128,-98.2679,87.5995,171.7383
C00560=1693.283,-149.465,-725.128,-97.5346,86.7171,172.4774
C00561=1693.196,-145.572,-725.128,-107.4295,88.0464,162.5825
C00562=1693.175,-142.266,-725.128,-88.6709,87.7083,-178.6711
C00563=1692.987,-139.610,-725.128,-87.3703,87.1067,-177.3762
C00564=1692.683,-134.034,-725.128,-81.6636,88.4704,-171.6696
C00565=1692.547,-129.592,-725.128,-74.2954,87.8229,-164.3071
C00566=1692.553,-124.530,-725.128,-103.6595,88.1495,166.3525
C00567=1692.491,-118.202,-725.128,-105.5789,86.5911,164.4503
C00568=1692.058,-113.505,-725.128,-95.2313,87.9662,174.7693
C00569=1692.024,-110.890,-725.128,-92.6243,88.5047,177.3762
C00570=1691.717,-106.496,-725.128,-94.0452,88.5162,175.9553
C00571=1691.849,-102.992,-725.128,-124.4063,87.7714,145.6114
C00572=1691.820,-99.398,-725.128,-120.5503,88.4073,149.4617
C00573=1691.518,-93.894,-725.128,-95.1854,88.7511,174.8151
C00574=1691.727,-90.920,-725.128,-136.1576,88.8657,133.8486
C00575=1691.521,-88.468,-725.128,-137.5442,89.6678,132.4563
C00576=1691.558,-83.592,-725.128,-117.2042,89.0433,152.7963
C00577=1691.757,-81.533,-725.128,-152.9052,88.4646,117.1011
C00578=1691.409,-75.937,-725.128,-107.2004,89.6163,162.8002
C00579=1691.267,-73.868,-725.128,-135.7508,89.3986,134.2497
C00580=1691.368,-69.992,-725.128,-139.8475,88.4818,130.1588
C00581=1691.497,-66.905,-725.128,-153.8162,88.5219,116.1958
C00582=1691.202,-62.642,-725.128,79.3546,89.7423,-10.6398
C00583=1690.949,-58.842,-725.128,-81.7037,89.8111,-171.7039
C00584=1691.102,-55.456,-725.128,-67.5116,89.7137,-157.5118
C00585=1691.059,-52.475,-725.128,67.3110,89.9085,-22.6891
C00586=1691.516,-46.324,-725.128,-173.9671,89.1006,96.0334
C00587=1691.447,-42.499,-725.128,-170.9075,88.8141,99.0930
C00588=1691.440,-37.363,-725.128,165.6306,88.8199,75.6246
C00589=1691.264,-34.202,-725.128,171.0680,89.0491,81.0677
C00590=1691.613,-29.953,-725.128,147.0267,88.5792,57.0207
C00591=1691.398,-25.866,-725.128,167.9167,88.6251,77.9108
C00592=1691.470,-22.076,-725.128,149.2211,88.2584,59.2094
C00593=1691.500,-18.159,-725.128,-177.5997,89.2496,92.4009
C00594=1691.331,-12.737,-725.128,129.0816,89.1522,39.0814
C00595=1691.544,-7.886,-725.128,95.7126,88.8542,5.7123
C00596=1691.477,-4.905,-725.128,155.2715,88.5620,65.2656
C00597=1691.865,-1.307,-725.128,31.2834,87.6911,-58.6937
C00598=1691.572,1.972,-725.128,125.9418,89.4730,35.9416
C00599=1691.649,6.374,-725.128,69.9466,89.3699,-20.0535
C00600=1691.423,10.417,-725.128,175.4052,89.0548,85.4050
C00601=1691.470,15.426,-725.128,179.2498,88.1037,89.2496
C00602=1691.943,16.520,-725.128,117.8688,88.0808,27.8572
C00603=1692.137,20.796,-725.128,127.7294,88.5792,37.7178
C00604=1691.889,23.766,-725.128,111.6522,88.3844,21.6406
C00605=1692.127,26.966,-725.128,146.2188,88.6938,56.2128
C00606=1692.577,31.210,-725.128,128.1706,88.9402,38.1647
C00607=1692.179,36.844,-725.128,161.4079,88.9631,71.4077
C00608=1692.102,39.325,-725.128,154.3147,89.3012,64.3145
C00609=1691.963,43.711,-725.128,86.1613,88.4990,-3.8388
C00610=1692.276,46.641,-725.128,130.0614,88.4933,40.0497
C00611=1692.298,50.614,-725.128,150.3670,87.8000,60.3496
C00612=1692.932,53.849,-725.128,150.6191,88.8657,60.6189
C00613=1692.972,58.007,-725.128,162.6512,87.6453,72.6395
C00614=1692.852,64.094,-725.128,136.9369,88.2469,46.9195
C00615=1692.938,66.408,-725.128,132.2386,88.4016,42.2269
C00616=1693.033,71.877,-725.128,147.3131,89.1407,57.3129
C00617=1692.911,73.086,-725.128,155.5866,87.9891,65.5692
C00618=1692.580,77.916,-725.128,88.6881,88.3959,-1.3120
C00619=1693.081,80.440,-725.128,148.7971,88.6251,58.7854
C00620=1692.999,84.182,-725.128,141.6981,88.3042,51.6807
C00621=1693.143,88.816,-725.128,138.8334,88.8657,48.8274
C00622=1692.709,92.833,-725.128,142.7868,89.0892,52.7808
C00623=1692.909,96.351,-725.128,157.5920,88.7397,67.5861
C00624=1693.248,98.029,-725.128,125.7756,88.3042,35.7640
C00625=1692.980,102.527,-725.128,150.2066,88.4188,60.2006
C00626=1693.040,105.070,-725.128,141.1939,88.5563,51.1823
C00627=1693.018,109.244,-725.128,124.9850,88.7511,34.9733
C00628=1693.458,111.504,-725.128,142.3513,88.4589,52.3396
C00629=1693.230,117.177,-725.128,126.6924,88.3672,36.6807
C00630=1693.513,120.828,-725.128,149.8170,89.5704,59.8167
C00631=1693.238,126.613,-725.128,115.7088,89.0949,25.7028
C00632=1693.802,128.159,-725.128,118.2928,89.6736,28.2926
C00633=1693.445,132.606,-725.128,80.8099,88.4646,-9.1845
C00634=1693.419,137.271,-725.128,81.0964,88.6136,-8.9037
C00635=1693.877,140.934,-725.128,128.9155,89.0548,38.9095
C00636=1693.696,145.465,-725.128,94.7213,88.6423,4.7211
C00637=1693.975,148.239,-725.128,159.9010,88.8485,69.8951
C00638=1694.009,152.974,-725.128,112.5919,89.0376,22.5917
C00639=1693.924,156.030,-725.128,167.8880,89.4387,77.8878
C00640=1693.898,160.064,-725.128,114.1045,89.4387,24.1043
C00641=1694.022,163.945,-725.128,122.5041,88.2526,32.4924
C00642=1694.158,168.032,-725.128,75.1606,88.8256,-14.8338
C00643=1694.079,171.275,-725.128,6.9156,89.0433,-83.0846
C00644=1694.151,176.630,-725.128,149.0950,89.5189,59.0948
C00645=1694.067,178.046,-725.128,23.2047,88.5277,-66.7839
C00646=1694.156,183.068,-725.128,95.2427,88.8313,5.2425
C00647=1694.232,186.390,-725.128,110.3287,88.7683,20.3228
C00648=1694.315,189.126,-725.128,74.8569,88.6308,-15.1375
C00649=1694.536,192.256,-725.128,100.8749,88.8084,10.8747
C00650=1694.451,196.132,-725.128,110.8673,89.3298,20.8671
C00651=1694.330,199.616,-725.128,165.1608,88.7798,75.1548
C00652=1694.507,203.227,-725.128,118.2814,89.0605,28.2811
C00653=1694.640,208.150,-725.128,131.0182,89.0433,41.0123
C00654=1694.478,210.745,-725.128,101.1843,88.8485,11.1841
C00655=1694.662,216.049,-725.128,35.7239,89.5704,-54.2762
C00656=1694.674,217.352,-725.128,107.7160,88.7683,17.7158
C00657=1694.625,221.604,-725.128,94.0109,87.7198,4.0107
C00658=1694.737,223.176,-725.128,91.0831,88.5563,1.0828
C00659=1694.916,226.335,-725.128,-175.4855,89.5017,94.5151
C00660=1694.902,227.683,-725.128,78.6842,89.2209,-11.3101
C00661=1694.903,231.089,-725.128,43.2640,89.1808,-46.7361
C00662=1694.957,234.305,-725.128,89.2152,83.2393,-0.7792
C00663=1695.307,235.674,-725.128,83.8867,78.5697,-5.9931
C00664=1695.280,235.559,-775.128,91.0258,73.5620,0.9854
C00665=1695.159,234.589,-775.128,96.9387,81.3199,6.8583
C00666=1694.773,231.875,-775.128,85.0498,86.4536,-4.9446
C00667=1694.791,229.585,-775.128,101.7057,88.1266,11.6997
C00668=1694.805,225.869,-775.128,-15.7276,88.7626,-105.7336
C00669=1694.794,223.920,-775.128,21.6749,89.6449,-68.3252
C00670=1694.786,222.595,-775.128,-155.6497,89.0605,114.3566
C00671=1694.646,218.486,-775.128,91.6732,89.1636,1.6730
C00672=1694.643,215.167,-775.128,30.8308,88.5391,-59.1636
C00673=1694.783,210.666,-775.128,81.9100,88.9688,-8.0901
C00674=1694.659,207.861,-775.128,129.4884,88.6365,39.4825
C00675=1694.726,204.677,-775.128,-96.6350,89.7423,173.3655
C00676=1694.675,201.200,-775.128,162.4564,89.5131,72.4562
C00677=1694.820,199.708,-775.128,58.9115,88.8027,-31.0829
C00678=1694.695,195.486,-775.128,122.6588,89.7538,32.6585
C00679=1694.396,191.453,-775.128,178.1841,89.4788,88.1839
C00680=1694.646,189.710,-775.128,154.9793,88.5334,64.9734
C00681=1694.371,185.227,-775.128,96.4058,88.8600,6.4056
C00682=1694.384,183.786,-775.128,112.1908,89.1980,22.1849
C00683=1694.617,180.852,-775.128,-45.9454,89.5762,-135.9456
C00684=1694.318,176.831,-775.128,-147.2730,88.7167,122.7390
C00685=1694.484,171.631,-775.128,179.9946,89.4387,89.9944
C00686=1694.549,170.698,-775.128,-170.5408,89.4673,99.4597
C00687=1694.315,166.804,-775.128,-25.0669,89.4501,-115.0671
C00688=1694.518,164.098,-775.128,-36.6291,89.7882,-126.6294
C00689=1694.521,160.609,-775.128,-46.5356,88.6995,-136.5415
C00690=1694.399,158.024,-775.128,128.4857,89.0949,38.4855
C00691=1694.100,155.305,-775.128,-166.8739,89.6048,103.1266
C00692=1694.580,150.859,-775.128,177.7257,88.8772,87.7255
C00693=1694.108,146.701,-775.128,28.7739,89.3241,-61.2205
C00694=1694.275,144.221,-775.128,8.6115,89.2439,-81.3886
C00695=1694.161,140.123,-775.128,-172.2769,89.7309,97.7236
C00696=1694.260,135.787,-775.128,178.6310,89.0433,88.6308
C00697=1694.433,132.332,-775.128,177.9377,89.0548,87.9375
C00698=1694.373,129.758,-775.128,-93.0483,89.3699,176.9522
C00699=1694.474,125.985,-775.128,-143.7035,87.6797,126.3200
C00700=1694.650,123.183,-775.128,-143.4800,87.9490,126.5377
C00701=1694.005,118.931,-775.128,90.1033,89.2954,0.1031
C00702=1694.023,115.371,-775.128,162.7658,88.8886,72.7656
C00703=1694.243,111.268,-775.128,151.3926,88.8944,61.3866
C00704=1694.349,107.562,-775.128,155.9877,89.5991,65.9875
C00705=1693.895,105.422,-775.128,146.2589,89.4616,56.2587
C00706=1694.008,100.769,-775.128,163.2471,89.0147,73.2469
C00707=1693.806,96.840,-775.128,72.0322,89.7538,-17.9679
C00708=1694.008,93.264,-775.128,150.2123,88.2355,60.2006
C00709=1693.666,89.449,-775.128,158.7780,89.4788,68.7778
C00710=1694.240,85.928,-775.128,142.6493,88.4589,52.6376
C00711=1693.879,81.183,-775.128,136.7191,88.8829,46.7132
C00712=1693.933,78.390,-775.128,-176.7861,89.2897,93.2145
C00713=1694.247,74.843,-775.128,158.1649,88.1782,68.1590
C00714=1693.474,71.802,-775.128,167.2922,86.8947,77.2748
C00715=1693.254,68.307,-775.128,139.9965,89.6392,49.9962
C00716=1693.596,64.411,-775.128,118.9002,87.3989,28.8770
C00717=1693.292,62.160,-775.128,162.0381,86.2817,72.0036
C00718=1694.049,58.527,-775.128,-179.8514,87.3416,90.1491
C00719=1693.009,56.555,-775.128,132.2902,89.1751,42.2842
C00720=1693.085,51.786,-775.128,153.6214,88.4646,63.6155
C00721=1693.390,48.460,-775.128,159.4770,89.2152,69.4768
C00722=1693.441,45.567,-775.128,124.1083,88.4131,34.0967
C00723=1692.734,41.255,-775.128,138.4094,86.9291,48.3690
C00724=1693.264,40.032,-775.128,127.2596,88.5391,37.2537
C00725=1692.977,36.970,-775.128,150.7681,88.3042,60.7564
C00726=1693.785,31.002,-775.128,164.5706,88.6537,74.5647
C00727=1693.321,29.063,-775.128,89.7481,89.0089,-0.2521
C00728=1693.681,25.546,-775.128,154.1944,88.0406,64.1770
C00729=1693.703,21.608,-775.128,143.5316,88.2068,53.5142
C00730=1692.607,17.413,-775.128,124.8876,89.4730,34.8874
C00731=1692.705,13.934,-775.128,148.4648,88.2813,58.4531
C00732=1692.582,10.554,-775.128,121.5529,88.5792,31.5470
C00733=1693.159,6.119,-775.128,159.9640,89.1121,69.9638
C00734=1692.987,2.306,-775.128,153.7303,87.9203,63.7129
C00735=1693.198,-0.580,-775.128,134.7310,89.0204,44.7250
C00736=1693.262,-3.471,-775.128,134.2955,89.9429,44.2953
C00737=1692.884,-7.851,-775.128,148.7627,87.8516,58.7396
C00738=1692.399,-12.054,-775.128,171.2914,88.6709,81.2912
C00739=1692.613,-14.656,-775.128,106.9597,88.5391,16.9538
C00740=1692.178,-17.963,-775.128,176.3965,88.1380,86.3963
C00741=1692.992,-22.676,-775.128,-179.2956,87.4791,90.7049
C00742=1693.367,-24.450,-775.128,-14.7422,86.5510,-104.7653
C00743=1692.140,-28.211,-775.128,136.7478,88.8027,46.7418
C00744=1691.974,-32.842,-775.128,128.2909,88.5964,38.2850
C00745=1691.865,-34.678,-775.128,142.8097,88.3959,52.8037
C00746=1693.154,-38.635,-775.128,102.6282,88.4704,12.6279
C00747=1692.169,-41.325,-775.128,-166.7479,87.8057,103.2584
C00748=1691.840,-47.021,-775.128,170.5065,88.3214,80.5005
C00749=1691.929,-50.154,-775.128,178.7742,88.9058,88.7740
C00750=1692.398,-53.005,-775.128,-175.2849,88.2584,94.7156
C00751=1693.146,-56.114,-775.128,169.9163,88.0979,79.9104
C00752=1692.493,-59.588,-775.128,154.2459,88.0235,64.2342
C00753=1692.138,-63.237,-775.128,-173.8697,88.6938,96.1308
C00754=1692.114,-66.379,-775.128,-177.9606,88.3959,92.0399
C00755=1692.843,-69.024,-775.128,161.0011,89.3814,71.0009
C00756=1691.957,-73.917,-775.128,173.5718,89.1636,83.5716
C00757=1691.814,-76.987,-775.128,168.9308,89.4272,78.9306
C00758=1692.733,-80.165,-775.128,-174.5229,88.5964,95.4776
C00759=1692.780,-84.946,-775.128,-154.5381,88.6308,115.4681
C00760=1692.187,-88.466,-775.128,-132.8861,89.3814,137.1202
C00761=1692.254,-91.320,-775.128,-165.5618,88.9459,104.4387
C00762=1692.211,-96.461,-775.128,175.6975,88.0922,85.6915
C00763=1692.013,-98.631,-775.128,-110.5178,89.3699,159.4828
C00764=1692.456,-102.953,-775.128,-173.0733,88.4131,96.9330
C00765=1692.753,-105.142,-775.128,-171.5664,87.8229,98.4398
C00766=1692.791,-109.369,-775.128,-163.5794,89.3986,106.4211
C00767=1692.367,-113.387,-775.128,-146.6199,89.3928,123.3807
C00768=1692.802,-116.780,-775.128,-134.4445,88.8313,135.5618
C00769=1692.428,-120.154,-775.128,-70.6743,88.6824,-160.6745
C00770=1692.995,-123.926,-775.128,-134.4846,88.1209,135.5331
C00771=1692.710,-127.569,-775.128,-108.5984,88.1667,161.4079
C00772=1692.717,-131.204,-775.128,-83.4169,88.1896,-173.4228
C00773=1693.137,-134.656,-775.128,-169.5668,87.8688,100.4395
C00774=1692.815,-138.280,-775.128,-133.1152,88.8772,136.8910
C00775=1693.104,-143.140,-775.128,-117.3131,87.6338,152.7047
C00776=1693.340,-146.610,-775.128,-153.1401,88.4532,116.8719
C00777=1693.161,-150.894,-775.128,-81.1021,88.7225,-171.1023
C00778=1693.309,-152.742,-775.128,-108.1114,88.5162,161.8949
C00779=1693.292,-156.731,-775.128,88.0521,87.2958,-1.9480
C00780=1693.053,-159.441,-775.128,17.0684,87.5021,-72.9203
C00781=1693.169,-161.869,-775.128,-81.6407,81.4917,-171.7326
C00782=1694.095,-162.262,-825.128,-78.7587,80.6208,-168.9079
C00783=1693.815,-161.320,-825.128,-91.1117,84.1331,178.8946
C00784=1693.694,-159.411,-825.128,-74.3470,84.7748,-164.4102
C00785=1693.835,-155.897,-825.128,81.3428,88.1151,-8.6516
C00786=1693.900,-152.136,-825.128,-65.4718,89.4673,-155.4720
C00787=1693.454,-149.528,-825.128,7.1161,89.3069,-82.8840
C00788=1693.684,-147.537,-825.128,-146.4308,89.4329,123.5698
C00789=1693.724,-142.723,-825.128,167.8479,88.6594,77.8477
C00790=1693.435,-138.200,-825.128,-139.9105,88.4188,130.1015
C00791=1693.263,-134.290,-825.128,-141.5778,88.9688,128.4227
C00792=1693.940,-128.596,-825.128,-152.8135,88.5792,117.1927
C00793=1694.179,-124.135,-825.128,178.6310,89.2954,88.6308
C00794=1694.185,-120.565,-825.128,0.6646,87.2270,-89.3298
C00795=1693.074,-118.342,-825.128,-128.7722,88.4532,141.2340
C00796=1693.871,-114.604,-825.128,0.9281,72.9031,-89.0261
C00797=1693.048,-112.378,-825.128,172.3342,88.4245,82.3340
C00798=1694.316,-109.326,-825.128,10.6799,86.8260,-79.3088
C00799=1693.190,-106.315,-825.128,-159.7979,88.2469,110.2084
C00800=1693.523,-102.267,-825.128,-173.4457,88.4073,96.5605
C00801=1693.270,-98.307,-825.128,170.7414,87.9261,80.7354
C00802=1693.937,-94.548,-825.128,166.0030,87.1526,75.9856
C00803=1693.556,-92.849,-825.128,155.1627,88.5620,65.1567
C00804=1694.360,-89.471,-825.128,-5.3628,88.3329,-95.3630
C00805=1693.850,-84.352,-825.128,177.9721,87.5995,87.9719
C00806=1693.997,-80.760,-825.128,-178.3273,87.0494,91.6732
C00807=1694.146,-75.961,-825.128,144.5629,86.9005,54.5283
C00808=1694.179,-75.053,-825.128,164.8170,87.6510,74.8053
C00809=1693.313,-72.193,-825.128,173.5202,88.7339,83.5200
C00810=1692.731,-67.375,-825.128,151.1061,88.0292,61.0944
C00811=1693.090,-63.308,-825.128,169.1887,87.5937,79.1827
C00812=1693.444,-58.799,-825.128,-179.8399,88.2985,90.1606
C00813=1694.003,-56.443,-825.128,152.9052,87.5880,62.8821
C00814=1694.156,-51.698,-825.128,178.9118,88.1552,88.9058
C00815=1693.179,-48.358,-825.128,-136.3868,87.8458,133.6309
C00816=1694.877,-45.134,-825.128,28.8369,86.4879,-61.1174
C00817=1694.494,-43.968,-825.128,1.7876,78.2488,-88.1782
C00818=1694.827,-39.536,-825.128,39.0413,89.5017,-50.9588
C00819=1694.546,-38.068,-825.128,146.0182,85.8634,55.9493
C00820=1694.047,-34.851,-825.128,144.4884,88.0120,54.4768
C00821=1693.287,-32.741,-825.128,143.1821,87.8573,53.1647
C00822=1693.637,-28.246,-825.128,-156.7383,87.0494,113.2852
C00823=1694.872,-25.166,-825.128,23.8293,87.1869,-66.1422
C00824=1694.206,-19.961,-825.128,160.4511,87.7141,70.4337
C00825=1693.988,-16.926,-825.128,166.2494,87.4161,76.2320
C00826=1695.007,-10.270,-825.128,135.1722,89.4329,45.1719
C00827=1693.494,-9.092,-825.128,129.9754,89.6105,39.9752
C00828=1693.831,-4.675,-825.128,152.1432,87.1812,62.1143
C00829=1693.821,-0.716,-825.128,147.3189,88.1896,57.3072
C00830=1695.030,4.742,-825.128,-174.0531,87.4161,95.9532
C00831=1694.269,8.958,-825.128,162.6455,89.1293,72.6453
C00832=1694.252,12.685,-825.128,70.2904,88.3099,-19.6982
C00833=1695.239,15.959,-825.128,25.1929,89.1694,-64.8072
C00834=1694.405,20.175,-825.128,169.9106,89.0433,79.9104
C00835=1695.082,24.566,-825.128,-3.6039,85.3477,-93.6155
C00836=1694.148,28.214,-825.128,163.7284,88.8256,73.7224
C00837=1694.455,31.493,-825.128,174.1963,86.9635,84.1904
C00838=1694.982,36.164,-825.128,165.1149,88.0120,75.1033
C00839=1695.288,39.974,-825.128,111.1480,89.6908,21.1478
C00840=1694.277,43.704,-825.128,145.2791,88.9058,55.2732
C00841=1695.018,45.352,-825.128,156.1825,87.5651,66.1651
C00842=1694.905,50.154,-825.128,151.4384,87.1067,61.4096
C00843=1694.322,51.954,-825.128,164.7712,88.1610,74.7595
C00844=1695.248,55.346,-825.128,136.6504,89.6908,46.6502
C00845=1694.732,60.073,-825.128,148.7455,89.1350,58.7396
C00846=1695.004,65.468,-825.128,-146.7459,87.8573,123.2718
C00847=1694.372,68.729,-825.128,177.6455,88.4818,87.6453
C00848=1694.675,72.104,-825.128,166.7020,88.1037,76.6961
C00849=1695.361,75.107,-825.128,-1.6959,85.3306,-91.7018
C00850=1695.030,79.516,-825.128,171.2055,89.2209,81.2053
C00851=1695.249,83.262,-825.128,-5.6722,79.7442,-95.7641
C00852=1695.418,86.450,-825.128,129.7176,88.3959,39.7059
C00853=1694.684,90.238,-825.128,153.8964,87.8917,63.8790
C00854=1694.504,92.614,-825.128,153.0714,88.8657,63.0654
C00855=1694.979,96.882,-825.128,-166.0431,88.6365,103.9574
C00856=1695.282,99.955,-825.128,-148.3101,86.6827,121.7306
C00857=1694.821,103.587,-825.128,-169.8017,89.3642,100.1988
C00858=1694.415,106.340,-825.128,149.0549,88.4131,59.0433
C00859=1695.139,109.931,-825.128,-173.6234,88.2698,96.3772
C00860=1694.795,113.963,-825.128,160.9438,88.4131,70.9379
C00861=1694.714,116.480,-825.128,154.8418,89.1350,64.8416
C00862=1694.885,120.619,-825.128,-18.2143,89.1407,-108.2202
C00863=1694.939,125.359,-825.128,-165.9343,88.4818,104.0663
C00864=1694.925,127.362,-825.128,165.4759,88.4933,75.4700
C00865=1695.358,131.443,-825.128,-10.1700,84.7576,-100.2103
C00866=1694.821,135.115,-825.128,-151.6103,89.1636,118.3902
C00867=1694.874,136.578,-825.128,-178.3216,88.7339,91.6789
C00868=1694.817,140.672,-825.128,-102.1927,88.7397,167.8078
C00869=1694.890,145.148,-825.128,148.4877,88.9746,58.4818
C00870=1694.568,148.641,-825.128,176.3621,88.7855,86.3619
C00871=1694.859,151.520,-825.128,113.3940,89.5074,23.3938
C00872=1694.992,157.338,-825.128,132.7886,89.6621,42.7884
C00873=1694.959,162.037,-825.128,-77.2690,89.1751,-167.2692
C00874=1694.902,165.267,-825.128,-178.5336,88.9516,91.4669
C00875=1694.742,172.042,-825.128,-175.2792,88.8886,94.7213
C00876=1695.262,176.077,-825.128,173.2624,89.3241,83.2564
C00877=1694.944,178.401,-825.128,168.8735,89.0662,78.8733
C00878=1694.964,182.387,-825.128,174.2250,89.0319,84.2190
C00879=1695.235,185.808,-825.128,125.9189,89.4845,35.9187
C00880=1695.185,189.761,-825.128,-2.1772,89.2610,-92.1774
C00881=1694.829,192.133,-825.128,-12.4675,89.5533,-102.4677
C00882=1694.887,196.365,-825.128,155.1111,88.7683,65.1051
C00883=1694.857,198.669,-825.128,156.7784,89.3871,66.7782
C00884=1694.754,201.884,-825.128,-55.3248,89.6507,-145.3250
C00885=1694.760,206.123,-825.128,-104.6564,89.5762,165.3441
C00886=1694.964,209.550,-825.128,-148.6424,88.9345,121.3581
C00887=1694.769,213.173,-825.128,-133.9632,88.0005,136.0545
C00888=1694.791,216.621,-825.128,20.0191,89.3126,-69.9810
C00889=1695.249,221.438,-825.128,-45.7564,87.3416,-135.7852
C00890=1694.882,222.542,-825.128,-156.0335,87.8745,113.9842
C00891=1695.078,225.878,-825.128,-2.6184,86.3905,-92.6243
C00892=1694.924,227.268,-825.128,174.7693,87.5422,84.7633
C00893=1694.725,231.410,-825.128,84.4597,87.0093,-5.5347
C00894=1694.952,233.477,-825.128,94.9276,84.0987,4.9045
C00895=1695.024,235.696,-825.128,91.8565,76.0372,1.8048
C00896=1793.675,208.803,-377.180,-3.9763,1.1573,-90.0002
C00897=1799.260,208.803,-377.522,-4.4175,-4.5722,-90.0002
C00898=1800.380,208.803,-377.828,-2.8877,0.1031,-90.0002
C00899=1804.392,208.803,-377.686,-2.2288,-4.5263,-90.0002
C00900=1805.238,208.803,-377.860,1.6100,-3.5122,-90.0002
C00901=1809.448,208.803,-378.127,-0.6703,-2.3835,-90.0002
C00902=1810.104,208.803,-378.034,0.3896,-1.1287,-90.0002
C00903=1815.541,208.803,-378.409,-2.3204,-3.5065,-90.0002
C00904=1816.234,208.803,-377.866,-5.5233,1.0198,-90.0002
C00905=1819.888,208.803,-378.043,-2.3262,-2.1428,-90.0002
C00906=1822.893,208.803,-378.295,-9.4996,2.1084,-90.0002
C00907=1825.029,208.803,-378.253,-5.2139,-2.6012,-90.0002
C00908=1828.890,208.803,-378.517,0.8021,-4.0794,-90.0002
C00909=1829.853,208.803,-378.619,-4.9560,1.2375,-90.0002
C00910=1834.434,208.803,-378.454,-0.5672,1.7131,-90.0002
C00911=1835.867,208.803,-378.912,-0.7734,-3.2486,-90.0002
C00912=1839.483,208.803,-378.247,-0.8708,1.1401,-90.0002
C00913=1841.644,208.803,-379.037,-3.8388,-1.9423,-90.0002
C00914=1844.398,208.803,-379.133,-3.1512,-2.5840,-90.0002
C00915=1849.534,208.803,-378.682,-2.0110,-2.1084,-90.0002
C00916=1850.191,208.803,-379.604,-1.5756,-4.0737,-90.0002
C00917=1854.259,208.803,-378.938,2.4866,-2.7616,-90.0002
C00918=1855.552,208.803,-378.611,-6.5202,1.4553,-90.0002
C00919=1859.933,208.803,-378.736,0.4755,-0.0401,-90.0002
C00920=1861.222,208.803,-378.901,0.3380,-1.9996,-90.0002
C00921=1865.407,208.803,-379.478,-0.1948,-1.4725,-90.0002
C00922=1869.854,208.803,-378.445,-1.9537,-2.1199,-90.0002
C00923=1870.486,208.803,-378.774,-6.9041,1.6959,-90.0002
C00924=1874.480,208.803,-380.418,-0.5328,-2.2746,-90.0002
C00925=1875.328,208.803,-379.048,-5.6035,-0.3093,-90.0002
C00926=1879.654,208.803,-379.098,-8.0901,1.8162,-90.0002
C00927=1880.591,208.803,-380.274,-7.1218,-0.6474,-90.0002
C00928=1884.581,208.803,-380.691,-5.6379,-3.1226,-90.0002
C00929=1888.675,208.803,-379.466,0.8938,-1.3865,-90.0002
C00930=1889.688,208.803,-379.350,-3.2715,0.5213,-90.0002
C00931=1893.936,208.803,-380.386,-3.3231,-2.7731,-90.0002
C00932=1894.825,208.803,-379.595,-1.4323,1.0026,-90.0002
C00933=1899.785,208.803,-380.090,-3.3861,0.9224,-90.0002
C00934=1900.882,208.803,-380.488,-3.9247,-1.8105,-90.0002
C00935=1904.672,208.803,-379.458,-4.8701,-2.6241,-90.0002
C00936=1906.870,208.803,-381.091,-3.2257,-1.7188,-90.0002
C00937=1909.764,208.803,-380.616,-3.7299,0.8136,-90.0002
C00938=1915.067,208.803,-379.839,-3.5007,-1.2605,-90.0002
C00939=1915.511,208.803,-381.230,-1.7761,-2.8476,-90.0002
C00940=1919.150,208.803,-378.820,-6.8067,1.3464,-90.0002
C00941=1921.049,208.803,-380.439,-3.3689,-2.3032,-90.0002
C00942=1924.399,208.803,-378.784,-4.1825,-1.0943,-90.0002
C00943=1926.037,208.803,-380.778,-1.6100,-0.2692,-90.0002
C00944=1929.785,208.803,-379.554,-7.5458,0.9912,-90.0002
C00945=1932.448,208.803,-380.390,-5.4545,1.9767,-90.0002
C00946=1934.473,208.803,-378.545,-10.8002,2.7158,-90.0002
C00947=1938.665,208.803,-379.236,-0.7161,1.1172,-90.0002
C00948=1939.972,208.803,-381.396,0.3724,1.7876,-90.0002
C00949=1944.120,208.803,-380.121,-1.2146,-1.7589,-90.0002
C00950=1945.329,208.803,-379.766,-3.6382,-1.4725,-90.0002
C00951=1949.489,208.803,-380.873,-4.6294,2.6527,-90.0002
C00952=1950.750,208.803,-379.083,-4.2513,1.4667,-90.0002
C00953=1954.631,208.803,-379.256,-2.8361,-0.6302,-90.0002
C00954=1956.191,208.803,-379.552,-6.4572,1.3292,-90.0002
C00955=1960.229,208.803,-379.116,-4.7211,-0.7906,-90.0002
C00956=1963.802,208.803,-381.137,-3.3747,-1.1459,-90.0002
C00957=1964.943,208.803,-378.752,-4.0508,-0.2922,-90.0002
C00958=1968.916,208.803,-380.754,-8.3365,1.4094,-90.0002
C00959=1970.139,208.803,-380.852,-3.2372,5.3514,-90.0002
C00960=1973.999,208.803,-380.062,-4.5550,2.9908,-90.0002
C00961=1975.489,208.803,-380.490,-5.8670,-1.0427,-90.0002
C00962=1979.540,208.803,-380.741,-2.2173,2.7501,-90.0002
C00963=1980.841,208.803,-379.906,-2.9392,1.4266,-90.0002
C00964=1984.548,208.803,-379.531,-2.4579,3.8961,-90.0002
C00965=1985.330,208.803,-377.747,-8.9094,5.0993,-90.0002
C00966=1989.044,208.803,-380.605,-1.1287,2.3835,-90.0002
C00967=1990.266,208.803,-377.667,-12.5993,-2.1772,-90.0002
C00968=1994.859,208.803,-379.373,-0.7333,2.0798,-90.0002
C00969=1995.564,208.803,-380.385,-1.7761,-2.6814,-90.0002
C00970=2000.220,208.803,-379.669,-3.9247,1.1573,-90.0002
C00971=2002.199,208.803,-379.938,-3.4090,4.0737,-90.0002
C00972=2005.140,208.803,-379.479,-0.6245,1.6959,-90.0002
C00973=2008.461,208.803,-378.774,-3.2486,4.9159,-90.0002
C00974=2010.347,208.803,-379.928,-5.5920,1.4725,-90.0002
C00975=2014.097,208.803,-380.402,-0.6474,-4.1424,-90.0002
C00976=2014.950,208.803,-379.359,-6.3770,2.9793,-90.0002
C00977=2018.830,208.803,-379.797,-2.7788,-0.3437,-90.0002
C00978=2019.895,208.803,-379.005,-2.9507,-1.1172,-90.0002
C00979=2023.913,208.803,-379.490,0.0458,3.5294,-90.0002
C00980=2024.936,208.803,-377.505,-0.5729,1.5355,-90.0002
C00981=2029.433,208.803,-379.336,-2.2803,-0.1890,-90.0002
C00982=2030.638,208.803,-379.630,-3.0137,0.6589,-90.0002
C00983=2035.518,208.803,-379.299,-2.1886,0.3953,-90.0002
C00984=2036.993,208.803,-379.866,-1.8048,-0.2463,-90.0002
C00985=2040.274,208.803,-379.622,-6.5832,1.0370,-90.0002
C00986=2041.009,208.803,-380.443,-3.5695,1.8105,-90.0002
C00987=2044.440,208.803,-379.299,-7.9354,2.8361,-90.0002
C00988=2049.189,208.803,-378.984,-1.4266,1.5011,-90.0002
C00989=2050.196,208.803,-379.315,-3.7815,1.8277,-90.0002
C00990=2054.969,208.803,-377.751,-2.7444,0.7734,-90.0002
C00991=2056.023,208.803,-380.655,-4.9388,1.0771,-90.0002
C00992=2059.833,208.803,-378.961,-0.3552,-2.7158,-90.0002
C00993=2060.654,208.803,-379.561,-5.3170,-1.8506,-90.0002
C00994=2064.797,208.803,-378.210,-6.5546,0.7734,-90.0002
C00995=2067.348,208.803,-379.260,-4.8644,2.4350,-90.0002
C00996=2070.116,208.803,-379.228,-5.0362,0.7104,-90.0002
C00997=2074.491,208.803,-378.624,-1.8563,0.9453,-90.0002
C00998=2075.255,208.803,-379.646,-2.3090,-1.7074,-90.0002
C00999=2079.276,208.803,-379.165,-1.8678,6.3254,-90.0002
C01000=2079.869,208.803,-377.136,0.2864,3.3174,-90.0002
C01001=2084.185,208.803,-378.837,-6.5489,6.5890,-90.0002
C01002=2085.181,208.803,-377.092,-15.1146,-4.5034,-90.0002
C01003=2088.476,208.803,-378.541,-0.5099,-2.6527,-90.0002
C01004=2090.558,208.803,-378.454,-0.8136,-1.4610,-90.0002
C01005=2094.855,208.803,-378.434,-1.9767,2.5095,-90.0002
C01006=2095.498,208.803,-377.348,-5.0420,2.7731,-90.0002
C01007=2099.183,208.803,-377.018,-5.0133,9.0756,-90.0002
C01008=2100.071,208.803,-379.064,0.3896,0.7505,-90.0002
C01009=2104.597,208.803,-377.906,-2.2459,4.0909,-90.0002
C01010=2105.223,208.803,-378.895,-0.3666,3.2028,-90.0002
C01011=2109.522,208.803,-378.143,-3.7586,3.0710,-90.0002
C01012=2110.162,208.803,-377.230,-6.7838,-0.4927,-90.0002
C01013=2113.905,208.803,-377.738,-4.1825,3.9133,-90.0002
C01014=2115.676,208.803,-377.544,-10.3934,3.7528,-90.0002
C01015=2116.867,208.803,-377.985,-1.3865,3.1111,-90.0002
C01016=2119.696,208.803,-377.935,-0.7391,3.1971,-90.0002
C01017=2121.655,208.803,-376.977,5.5634,-4.5550,-90.0002
C01018=2124.496,208.803,-378.352,0.5042,2.9163,-90.0002
C01019=2125.342,208.803,-378.091,-4.5378,3.7643,-90.0002
C01020=2130.096,208.803,-377.169,-2.8246,2.5668,-90.0002
C01021=2132.447,208.803,-376.804,-1.0599,1.0943,-90.0002
C01022=2135.245,208.803,-377.232,-0.1317,-5.8957,-90.0002
C01023=2136.828,208.803,-376.772,-6.2509,3.6268,-90.0002
C01024=2139.609,208.803,-377.333,-0.9339,6.0561,-90.0002
C01025=2140.815,208.803,-377.552,-2.3777,0.3953,-90.0002
C01026=2144.185,208.803,-377.207,-1.2834,1.1802,-90.0002
C01027=2145.974,208.803,-377.282,-2.2746,-0.1260,-90.0002
C01028=2149.228,208.803,-377.060,-4.0393,3.3231,-90.0002
C01029=2150.114,208.803,-377.167,0.8537,1.7647,-90.0002
C01030=2151.355,208.803,-376.906,2.0397,1.1631,-90.0002
C01031=2154.711,208.803,-377.071,-4.0450,-1.1172,-90.0002
C01032=2155.831,208.803,-377.169,1.6959,-2.1084,-90.0002
C01033=2158.437,208.803,-377.483,-3.0080,2.8304,-90.0002
C01034=2159.759,208.803,-376.882,-0.7333,0.3552,-90.0002
C01035=2160.644,208.803,-376.885,-1.0026,5.4373,-90.0002
C01036=2163.605,208.803,-376.753,-1.5699,1.2375,-90.0002
C01037=2165.435,208.803,-376.757,-1.3521,0.5557,-90.0002
C01038=2165.872,208.803,-377.076,15.1719,-0.0744,-90.0002
C01039=2169.376,208.803,-377.119,1.8334,-2.8361,-90.0002
C01040=2170.477,208.803,-376.733,-3.6325,4.4175,-90.0002
C01041=2171.900,208.803,-377.095,-4.3315,4.4117,-90.0002
C01042=2174.172,208.803,-376.883,5.5748,-0.4239,-90.0002
C01043=2175.393,208.803,-377.068,1.7131,2.0397,-90.0002
C01044=2177.857,208.803,-376.746,0.5729,4.4805,-90.0002
C01045=2180.118,208.803,-376.259,-1.5469,1.4954,-90.0002
C01046=2183.652,208.803,-377.007,3.8044,-0.1546,-90.0002
C01047=2185.084,208.803,-376.532,-4.6638,2.0454,-90.0002
C01048=2186.051,158.803,-375.227,0.3838,-0.7505,-90.0002
C01049=2184.581,158.803,-375.378,-2.5038,6.5202,-90.0002
C01050=2180.434,158.803,-376.133,1.5011,4.8529,-90.0002
C01051=2179.702,158.803,-376.823,-1.5584,6.1134,-90.0002
C01052=2175.880,158.803,-376.616,-1.2032,5.8842,-90.0002
C01053=2174.439,158.803,-377.104,-1.9709,3.0653,-90.0002
C01054=2173.422,158.803,-377.056,-0.9396,5.8785,-90.0002
C01055=2170.660,158.803,-376.721,1.7074,3.5580,-90.0002
C01056=2170.235,158.803,-376.503,0.9912,0.4870,-90.0002
C01057=2169.305,158.803,-377.176,-0.9568,3.0137,-90.0002
C01058=2167.225,158.803,-376.867,-0.7563,5.3915,-90.0002
C01059=2165.148,158.803,-376.924,-1.9079,2.8246,-90.0002
C01060=2164.554,158.803,-377.230,0.0802,2.4465,-90.0002
C01061=2160.888,158.803,-377.453,0.1375,2.6356,-90.0002
C01062=2160.115,158.803,-377.533,-2.6527,2.6699,-90.0002
C01063=2155.393,158.803,-377.509,-0.3781,1.5870,-90.0002
C01064=2154.510,158.803,-378.041,0.6359,3.0710,-90.0002
C01065=2149.754,158.803,-377.602,-0.9854,0.5786,-90.0002
C01066=2148.910,158.803,-377.636,-2.7387,4.8987,-90.0002
C01067=2145.138,158.803,-378.176,-4.2055,5.3743,-90.0002
C01068=2143.685,158.803,-377.478,0.3724,2.8361,-90.0002
C01069=2140.371,158.803,-378.907,-1.6042,4.5722,-90.0002
C01070=2139.559,158.803,-377.848,-1.9537,2.3835,-90.0002
C01071=2135.153,158.803,-379.008,-4.1367,1.4152,-90.0002
C01072=2134.071,158.803,-378.324,-0.9797,1.8277,-90.0002
C01073=2130.265,158.803,-379.200,-4.0393,3.1799,-90.0002
C01074=2129.504,158.803,-378.851,-1.6673,4.7612,-90.0002
C01075=2124.870,158.803,-378.184,-0.2750,3.1111,-90.0002
C01076=2124.336,158.803,-379.532,-1.5240,2.6871,-90.0002
C01077=2119.547,158.803,-378.739,-0.3896,1.5756,-90.0002
C01078=2118.678,158.803,-379.070,0.4755,3.6898,-90.0002
C01079=2114.948,158.803,-379.673,-0.0343,3.2028,-90.0002
C01080=2114.156,158.803,-379.062,-1.9251,5.3858,-90.0002
C01081=2109.806,158.803,-379.761,-2.6757,3.0825,-90.0002
C01082=2108.644,158.803,-379.351,-2.3319,1.4610,-90.0002
C01083=2105.025,158.803,-379.781,-6.2853,2.7731,-90.0002
C01084=2104.038,158.803,-380.327,-0.6703,-0.7276,-90.0002
C01085=2099.906,158.803,-379.049,-0.7104,-0.6531,-90.0002
C01086=2099.307,158.803,-379.441,-1.1860,1.5297,-90.0002
C01087=2094.144,158.803,-379.808,-5.1337,2.4579,-90.0002
C01088=2093.296,158.803,-380.550,-2.8132,1.3235,-90.0002
C01089=2089.469,158.803,-380.757,-2.6012,1.4209,-90.0002
C01090=2087.431,158.803,-380.036,-0.0744,1.7360,-90.0002
C01091=2085.451,158.803,-380.723,-2.5668,2.2517,-90.0002
C01092=2084.030,158.803,-380.832,0.9854,3.0595,-90.0002
C01093=2080.035,158.803,-379.737,-4.1482,3.4835,-90.0002
C01094=2079.484,158.803,-381.390,-1.5126,1.4896,-90.0002
C01095=2074.709,158.803,-380.984,-1.3178,3.3804,-90.0002
C01096=2074.032,158.803,-381.188,-4.7555,4.8586,-90.0002
C01097=2070.281,158.803,-379.963,0.3609,0.9797,-90.0002
C01098=2068.312,158.803,-381.360,-2.2001,-0.9625,-90.0002
C01099=2065.267,158.803,-380.813,-1.2605,0.2807,-90.0002
C01100=2064.509,158.803,-381.262,-6.3541,4.0221,-90.0002
C01101=2060.241,158.803,-381.026,-2.0225,1.0026,-90.0002
C01102=2059.134,158.803,-380.368,-1.4037,5.4774,-90.0002
C01103=2055.026,158.803,-381.956,-3.0767,0.8021,-90.0002
C01104=2053.840,158.803,-380.488,1.3349,-0.8422,-90.0002
C01105=2050.032,158.803,-380.980,-3.3804,3.1627,-90.0002
C01106=2049.382,158.803,-381.344,-2.3319,-3.1226,-90.0002
C01107=2046.013,158.803,-381.188,1.4037,-1.4667,-90.0002
C01108=2044.577,158.803,-381.354,-4.9274,-0.4239,-90.0002
C01109=2043.336,158.803,-381.945,-7.4541,3.8445,-90.0002
C01110=2040.178,158.803,-380.743,-2.8533,4.0508,-90.0002
C01111=2038.975,158.803,-381.913,1.1229,-2.6184,-90.0002
C01112=2034.929,158.803,-380.462,-4.2628,2.6356,-90.0002
C01113=2034.396,158.803,-381.111,-5.0477,2.3262,-90.0002
C01114=2033.042,158.803,-381.957,-1.9938,0.3208,-90.0002
C01115=2029.727,158.803,-381.029,-1.1344,-0.6245,-90.0002
C01116=2029.341,158.803,-382.295,-0.6703,-1.2146,-90.0002
C01117=2025.552,158.803,-382.046,0.2750,0.3437,-90.0002
C01118=2024.557,158.803,-382.231,0.1948,1.3349,-90.0002
C01119=2020.436,158.803,-380.874,-4.1023,0.4239,-90.0002
C01120=2019.721,158.803,-381.449,-2.0225,0.4526,-90.0002
C01121=2016.222,158.803,-381.350,-6.8411,0.4354,-90.0002
C01122=2014.762,158.803,-382.372,1.1401,-0.9167,-90.0002
C01123=2012.972,158.803,-381.143,-0.7276,0.7276,-90.0002
C01124=2010.802,158.803,-382.149,1.1860,-1.7246,-90.0002
C01125=2009.611,158.803,-380.843,-1.4896,-0.3724,-90.0002
C01126=2005.829,158.803,-382.603,-6.7036,0.2864,-90.0002
C01127=2004.633,158.803,-380.983,-3.0710,-0.6703,-90.0002
C01128=2003.963,158.803,-382.004,-1.1115,-0.3093,-90.0002
C01129=1999.793,158.803,-381.636,-1.5985,-1.7532,-90.0002
C01130=1998.672,158.803,-380.959,-5.4029,1.6042,-90.0002
C01131=1995.138,158.803,-381.995,3.3288,0.0802,-90.0002
C01132=1994.325,158.803,-382.180,0.7391,1.3865,-90.0002
C01133=1991.038,158.803,-381.239,-0.8594,-0.7677,-90.0002
C01134=1990.264,158.803,-381.404,-2.3491,-1.2204,-90.0002
C01135=1987.335,158.803,-381.891,4.6065,-0.2406,-90.0002
C01136=1985.001,158.803,-381.232,-5.6092,0.9396,-90.0002
C01137=1983.940,158.803,-382.412,0.9797,0.2635,-90.0002
C01138=1979.773,158.803,-381.409,-1.4381,2.3147,-90.0002
C01139=1977.450,158.803,-382.265,-5.4602,1.7647,-90.0002
C01140=1974.887,158.803,-381.518,-6.8067,2.3204,-90.0002
C01141=1973.704,158.803,-381.791,1.4152,4.2341,-90.0002
C01142=1971.251,158.803,-381.745,1.3579,0.0916,-90.0002
C01143=1969.658,158.803,-382.264,0.2807,2.8017,-90.0002
C01144=1968.961,158.803,-381.733,-3.8560,-5.1508,-90.0002
C01145=1965.016,158.803,-382.561,-1.4782,-0.9167,-90.0002
C01146=1964.109,158.803,-382.767,-5.5290,1.7647,-90.0002
C01147=1960.588,158.803,-381.399,-3.2601,0.6474,-90.0002
C01148=1959.256,158.803,-381.765,-1.9365,3.3804,-90.0002
C01149=1956.483,158.803,-381.654,-2.0397,2.2116,-90.0002
C01150=1954.915,158.803,-382.719,-1.8048,0.7964,-90.0002
C01151=1951.244,158.803,-381.753,1.0084,6.3025,-90.0002
C01152=1949.542,158.803,-380.959,-3.6497,0.8136,-90.0002
C01153=1948.564,158.803,-382.650,3.5924,0.9568,-90.0002
C01154=1944.845,158.803,-382.989,-4.8701,2.4121,-90.0002
C01155=1943.650,158.803,-382.854,-0.1375,2.2975,-90.0002
C01156=1940.249,158.803,-382.312,0.3896,0.5500,-90.0002
C01157=1939.985,158.803,-383.091,-1.6386,5.6665,-90.0002
C01158=1936.858,158.803,-382.264,-5.0534,1.4266,-90.0002
C01159=1935.151,158.803,-382.287,0.3495,0.8708,-90.0002
C01160=1931.866,158.803,-382.106,-3.6039,3.0309,-90.0002
C01161=1929.856,158.803,-383.067,-2.8762,-1.3063,-90.0002
C01162=1928.280,158.803,-381.657,-0.8880,-1.9194,-90.0002
C01163=1924.931,158.803,-383.328,-2.1772,-0.2635,-90.0002
C01164=1924.145,158.803,-382.535,-5.6149,2.5783,-90.0002
C01165=1920.513,158.803,-382.142,-3.4205,-0.4182,-90.0002
C01166=1919.312,158.803,-382.391,-1.7818,-2.2173,-90.0002
C01167=1914.493,158.803,-382.086,-2.4178,1.8048,-90.0002
C01168=1914.330,158.803,-382.749,2.4751,-1.2891,-90.0002
C01169=1911.180,158.803,-382.835,-2.0053,2.8304,-90.0002
C01170=1909.902,158.803,-381.762,-7.2880,-0.5443,-90.0002
C01171=1906.067,158.803,-382.842,1.3235,-0.4583,-90.0002
C01172=1905.011,158.803,-382.641,-3.5867,-1.5928,-90.0002
C01173=1900.583,158.803,-382.797,-1.7818,-1.6042,-90.0002
C01174=1899.788,158.803,-382.172,-1.9308,-0.8250,-90.0002
C01175=1895.760,158.803,-381.886,-4.2341,0.5500,-90.0002
C01176=1894.594,158.803,-382.626,-3.4663,-1.3120,-90.0002
C01177=1892.203,158.803,-382.091,-3.9648,-1.3750,-90.0002
C01178=1890.022,158.803,-381.622,-1.8506,-2.6986,-90.0002
C01179=1888.748,158.803,-381.651,-4.1596,-4.5034,-90.0002
C01180=1885.598,158.803,-381.584,1.1745,3.9705,-90.0002
C01181=1884.835,158.803,-382.372,-4.8472,0.0401,-90.0002
C01182=1883.408,158.803,-381.827,-4.6065,-2.1772,-90.0002
C01183=1879.477,158.803,-382.180,-1.5068,-0.9854,-90.0002
C01184=1878.971,158.803,-381.181,-0.8766,-2.4006,-90.0002
C01185=1874.971,158.803,-381.141,-2.2803,-0.6703,-90.0002
C01186=1874.190,158.803,-382.209,-0.2521,-2.4923,-90.0002
C01187=1870.334,158.803,-380.407,-3.4721,-0.0114,-90.0002
C01188=1869.469,158.803,-381.574,-4.6982,-0.2922,-90.0002
C01189=1865.393,158.803,-380.688,-3.3632,-3.3174,-90.0002
C01190=1864.744,158.803,-380.585,1.1974,0.3838,-90.0002
C01191=1862.140,158.803,-382.096,-5.9129,-4.6123,-90.0002
C01192=1860.194,158.803,-380.808,-2.2803,-2.7559,-90.0002
C01193=1859.245,158.803,-381.117,-0.9568,-0.2578,-90.0002
C01194=1855.289,158.803,-380.403,0.1890,-4.6581,-90.0002
C01195=1854.730,158.803,-380.374,-0.3437,-1.0657,-90.0002
C01196=1850.109,158.803,-380.039,-5.5061,-1.8621,-90.0002
C01197=1849.392,158.803,-380.126,-3.5752,-5.5920,-90.0002
C01198=1845.224,158.803,-379.567,-3.4893,0.8651,-90.0002
C01199=1844.348,158.803,-379.823,-5.8613,-1.3464,-90.0002
C01200=1840.144,158.803,-379.377,-0.4297,-2.7673,-90.0002
C01201=1839.522,158.803,-380.278,-4.2055,-3.9247,-90.0002
C01202=1835.275,158.803,-379.806,-4.3315,-0.8021,-90.0002
C01203=1834.424,158.803,-380.477,-1.0943,-3.9018,-90.0002
C01204=1830.269,158.803,-379.575,2.5783,-1.3579,-90.0002
C01205=1828.414,158.803,-378.766,-2.9564,-0.8766,-90.0002
C01206=1824.701,158.803,-378.747,-2.4751,-0.7849,-90.0002
C01207=1823.852,158.803,-379.628,-2.8132,0.0000,-90.0002
C01208=1819.681,158.803,-379.287,-1.6959,-3.5981,-90.0002
C01209=1818.352,158.803,-379.128,0.0401,-1.6100,-90.0002
C01210=1815.253,158.803,-378.511,0.4870,-2.3777,-90.0002
C01211=1814.405,158.803,-378.620,-3.3403,-0.9969,-90.0002
C01212=1810.294,158.803,-378.646,-0.7505,-3.3804,-90.0002
C01213=1808.202,158.803,-378.307,-1.5584,-0.4870,-90.0002
C01214=1805.361,158.803,-378.314,-0.3552,-4.2226,-90.0002
C01215=1803.949,158.803,-378.205,0.6302,-0.5271,-90.0002
C01216=1800.699,158.803,-378.463,-2.3892,-6.8869,-90.0002
C01217=1799.347,158.803,-377.779,-0.0515,-2.6470,-90.0002
C01218=1795.852,158.803,-377.554,0.3036,3.2945,-90.0002
C01219=1794.744,108.803,-377.373,-1.8277,-6.3655,-90.0002
C01220=1795.283,108.803,-377.674,-0.6760,-6.0045,-90.0002
C01221=1798.437,108.803,-378.634,-4.1138,-7.5802,-90.0002
C01222=1799.550,108.803,-378.136,-4.7784,-1.9881,-90.0002
C01223=1804.214,108.803,-378.939,1.8735,-6.7150,-90.0002
C01224=1805.330,108.803,-378.791,-0.8651,-4.0107,-90.0002
C01225=1809.117,108.803,-378.677,-4.1539,-2.8762,-90.0002
C01226=1810.050,108.803,-379.328,1.6673,-2.9679,-90.0002
C01227=1812.965,108.803,-379.523,0.2062,-3.3976,-90.0002
C01228=1814.493,108.803,-379.691,-1.9079,-6.2681,-90.0002
C01229=1818.922,108.803,-379.770,-1.5870,-4.2857,-90.0002
C01230=1819.903,108.803,-380.055,0.7047,-3.7929,-90.0002
C01231=1823.323,108.803,-379.996,0.3437,-0.4927,-90.0002
C01232=1824.695,108.803,-379.868,-1.7704,-3.6898,-90.0002
C01233=1829.240,108.803,-380.232,0.3380,-1.6329,-90.0002
C01234=1830.010,108.803,-380.649,0.5385,-0.3666,-90.0002
C01235=1832.538,108.803,-380.599,-1.8277,-4.2169,-90.0002
C01236=1834.830,108.803,-380.317,-1.8048,-4.3143,-90.0002
C01237=1839.193,108.803,-380.576,-2.4006,-3.4549,-90.0002
C01238=1840.213,108.803,-380.897,-1.9537,-2.5840,-90.0002
C01239=1843.785,108.803,-381.601,-0.4927,-4.5435,-90.0002
C01240=1845.473,108.803,-381.963,0.6016,-4.7899,-90.0002
C01241=1845.654,108.803,-381.932,-0.5271,-2.5152,-90.0002
C01242=1849.452,108.803,-381.793,-3.5236,1.0485,-90.0002
C01243=1850.223,108.803,-381.879,-0.6589,-0.5614,-90.0002
C01244=1851.727,108.803,-382.056,1.8964,-3.1512,-90.0002
C01245=1854.851,108.803,-382.035,-2.4694,-1.1000,-90.0002
C01246=1855.709,108.803,-381.449,0.4640,-3.3747,-90.0002
C01247=1859.761,108.803,-382.440,0.1718,-1.8162,-90.0002
C01248=1860.563,108.803,-382.517,-3.0939,-2.5095,-90.0002
C01249=1861.767,108.803,-381.993,-1.2776,-5.5519,-90.0002
C01250=1864.201,108.803,-382.523,-0.0572,-1.9365,-90.0002
C01251=1866.076,108.803,-382.567,-2.9048,0.7849,-90.0002
C01252=1869.525,108.803,-382.551,-1.8907,-2.0912,-90.0002
C01253=1870.289,108.803,-382.429,-1.3693,-2.8533,-90.0002
C01254=1875.008,108.803,-382.747,-0.9568,0.1890,-90.0002
C01255=1876.033,108.803,-382.632,-5.3113,0.5385,-90.0002
C01256=1879.817,108.803,-382.586,-1.5699,-1.5527,-90.0002
C01257=1880.355,108.803,-382.620,4.0737,-4.7612,-90.0002
C01258=1884.434,108.803,-383.154,-2.3262,-2.9908,-90.0002
C01259=1885.347,108.803,-383.047,-2.2517,-2.7043,-90.0002
C01260=1889.287,108.803,-383.436,0.7276,-0.3724,-90.0002
C01261=1890.720,108.803,-382.878,-3.6153,1.8391,-90.0002
C01262=1894.258,108.803,-383.326,0.4469,-1.4896,-90.0002
C01263=1896.162,108.803,-382.987,-0.8365,-2.2918,-90.0002
C01264=1899.897,108.803,-383.389,-0.0916,-1.1860,-90.0002
C01265=1900.916,108.803,-383.403,-2.5668,-0.3036,-90.0002
C01266=1905.062,108.803,-383.932,-2.0454,-1.2547,-90.0002
C01267=1905.704,108.803,-383.234,0.0744,2.2861,-90.0002
C01268=1908.888,108.803,-383.727,-1.3865,0.2234,-90.0002
C01269=1909.936,108.803,-383.142,-5.2826,-0.1432,-90.0002
C01270=1914.697,108.803,-383.117,-4.8013,-0.0515,-90.0002
C01271=1916.137,108.803,-383.399,-0.2234,3.5867,-90.0002
C01272=1919.285,108.803,-383.089,-2.9965,0.9797,-90.0002
C01273=1919.909,108.803,-383.805,0.6130,-1.5699,-90.0002
C01274=1924.508,108.803,-383.980,-0.5672,-2.4923,-90.0002
C01275=1925.664,108.803,-383.772,-5.1852,7.1848,-90.0002
C01276=1929.305,108.803,-383.905,0.8938,0.4068,-90.0002
C01277=1930.380,108.803,-383.246,-2.7501,-2.9220,-90.0002
C01278=1934.724,108.803,-383.324,1.9423,0.7276,-90.0002
C01279=1936.137,108.803,-383.827,-2.0626,0.3838,-90.0002
C01280=1939.690,108.803,-383.432,0.6703,3.0481,-90.0002
C01281=1940.791,108.803,-384.389,1.6902,-2.6241,-90.0002
C01282=1944.547,108.803,-383.113,0.5557,-0.0458,-90.0002
C01283=1945.223,108.803,-383.374,6.7666,6.1936,-90.0002
C01284=1949.590,108.803,-383.510,0.8651,0.5099,-90.0002
C01285=1950.926,108.803,-383.959,2.2689,3.3403,-90.0002
C01286=1955.180,108.803,-383.004,1.3063,-2.4064,-90.0002
C01287=1956.475,108.803,-383.052,-3.9476,1.2318,-90.0002
C01288=1959.975,108.803,-383.156,0.5614,1.1917,-90.0002
C01289=1960.732,108.803,-383.011,-5.1909,0.4297,-90.0002
C01290=1964.501,108.803,-383.214,-0.1833,5.3915,-90.0002
C01291=1966.277,108.803,-383.011,1.2547,-0.8365,-90.0002
C01292=1969.836,108.803,-383.713,0.4469,4.1367,-90.0002
C01293=1970.819,108.803,-383.013,-0.4068,-0.2807,-90.0002
C01294=1974.872,108.803,-383.569,-0.2578,2.1371,-90.0002
C01295=1975.784,108.803,-383.326,-1.4152,-0.5156,-90.0002
C01296=1980.213,108.803,-383.311,-2.7387,1.4839,-90.0002
C01297=1980.915,108.803,-383.012,-1.1631,0.1145,-90.0002
C01298=1984.723,108.803,-382.898,-4.4289,0.0687,-90.0002
C01299=1985.767,108.803,-383.269,0.3323,1.1401,-90.0002
C01300=1990.375,108.803,-382.755,3.6325,-1.9824,-90.0002
C01301=1991.153,108.803,-382.934,-2.5725,1.2318,-90.0002
C01302=1994.951,108.803,-382.911,-1.9881,1.1172,-90.0002
C01303=1995.784,108.803,-382.933,-0.3265,1.0313,-90.0002
C01304=1999.864,108.803,-382.796,-2.6356,1.1688,-90.0002
C01305=2000.574,108.803,-382.692,-0.7333,-1.4610,-90.0002
C01306=2004.866,108.803,-383.199,-0.5443,2.0569,-90.0002
C01307=2007.056,108.803,-383.284,0.9797,-1.3579,-90.0002
C01308=2009.897,108.803,-382.958,0.7792,2.4408,-90.0002
C01309=2010.997,108.803,-382.499,3.7471,1.9709,-90.0002
C01310=2014.605,108.803,-383.059,1.2776,0.9110,-90.0002
C01311=2015.715,108.803,-382.609,4.2226,2.5783,-90.0002
C01312=2019.736,108.803,-382.900,-5.3628,1.3407,-90.0002
C01313=2020.984,108.803,-383.145,-0.6990,3.3059,-90.0002
C01314=2024.713,108.803,-382.436,-2.3491,1.9824,-90.0002
C01315=2025.539,108.803,-382.856,-4.1596,2.3262,-90.0002
C01316=2029.502,108.803,-382.819,-6.2223,-1.5355,-90.0002
C01317=2031.463,108.803,-382.252,-4.8071,2.6012,-90.0002
C01318=2034.505,108.803,-382.390,-7.9354,3.3174,-90.0002
C01319=2035.972,108.803,-382.159,-4.0049,0.0572,-90.0002
C01320=2039.787,108.803,-382.187,-4.6925,1.6673,-90.0002
C01321=2040.832,108.803,-383.110,1.1287,-1.4209,-90.0002
C01322=2044.710,108.803,-382.573,-1.0084,-0.2807,-90.0002
C01323=2045.413,108.803,-382.211,-3.9247,5.3113,-90.0002
C01324=2049.724,108.803,-382.574,3.5523,-0.7505,-90.0002
C01325=2050.256,108.803,-382.121,0.5557,0.9625,-90.0002
C01326=2051.382,108.803,-381.752,0.2349,2.9392,-90.0002
C01327=2054.010,108.803,-382.504,-0.2864,1.7761,-90.0002
C01328=2055.568,108.803,-382.106,-0.5729,0.8365,-90.0002
C01329=2059.213,108.803,-382.574,-1.4725,0.1604,-90.0002
C01330=2060.480,108.803,-382.559,1.3750,1.2605,-90.0002
C01331=2063.614,108.803,-382.682,-1.1344,-3.3231,-90.0002
C01332=2065.104,108.803,-382.001,2.0741,2.5840,-90.0002
C01333=2066.757,108.803,-382.084,-0.3896,-0.3552,-90.0002
C01334=2069.094,108.803,-382.215,-1.8850,7.1275,-90.0002
C01335=2070.547,108.803,-382.302,3.1684,-0.1375,-90.0002
C01336=2072.932,108.803,-382.198,-5.3456,6.0676,-90.0002
C01337=2074.436,108.803,-381.761,-3.8273,5.7123,-90.0002
C01338=2076.512,108.803,-382.087,-2.5783,-0.8422,-90.0002
C01339=2079.098,108.803,-382.350,-7.5343,11.0007,-90.0002
C01340=2080.360,108.803,-381.448,-4.1023,5.3113,-90.0002
C01341=2081.878,108.803,-382.094,-5.9988,1.6558,-90.0002
C01342=2084.796,108.803,-381.398,-4.5664,1.5297,-90.0002
C01343=2085.871,108.803,-381.549,-0.9110,4.8586,-90.0002
C01344=2089.136,108.803,-381.599,-1.7933,1.8964,-90.0002
C01345=2090.023,108.803,-381.861,1.0542,-0.7219,-90.0002
C01346=2093.346,108.803,-381.946,-1.8506,-6.1363,-90.0002
C01347=2094.329,108.803,-381.454,-3.3518,6.7265,-90.0002
C01348=2098.156,108.803,-381.345,0.3781,0.6703,-90.0002
C01349=2100.038,108.803,-380.948,-2.0626,0.3151,-90.0002
C01350=2103.365,108.803,-380.867,-1.9938,2.9106,-90.0002
C01351=2105.270,108.803,-380.870,-1.9996,4.4060,-90.0002
C01352=2108.636,108.803,-380.785,0.0000,4.8071,-90.0002
C01353=2110.171,108.803,-380.810,-1.7704,2.5382,-90.0002
C01354=2114.318,108.803,-380.633,-2.2116,2.6356,-90.0002
C01355=2114.968,108.803,-380.419,1.3750,3.2257,-90.0002
C01356=2118.593,108.803,-380.570,-2.3090,5.3628,-90.0002
C01357=2119.933,108.803,-380.360,0.4870,3.1283,-90.0002
C01358=2123.489,108.803,-379.750,-4.8644,4.3430,-90.0002
C01359=2124.467,108.803,-379.731,1.0943,4.3487,-90.0002
C01360=2128.885,108.803,-379.930,0.4354,2.6585,-90.0002
C01361=2129.833,108.803,-379.787,-0.6703,3.3689,-90.0002
C01362=2134.538,108.803,-379.118,-0.8307,2.3892,-90.0002
C01363=2135.914,108.803,-379.359,-1.7188,3.2486,-90.0002
C01364=2139.422,108.803,-379.144,-1.4152,4.9388,-90.0002
C01365=2140.335,108.803,-378.952,0.2578,3.0137,-90.0002
C01366=2142.949,108.803,-378.572,0.6016,4.6352,-90.0002
C01367=2144.844,108.803,-378.971,-2.7788,5.6207,-90.0002
C01368=2148.346,108.803,-378.603,-0.2750,4.1596,-90.0002
C01369=2149.570,108.803,-378.482,0.8708,2.8189,-90.0002
C01370=2153.470,108.803,-378.271,-1.5584,6.2337,-90.0002
C01371=2155.140,108.803,-378.024,-1.6443,3.4778,-90.0002
C01372=2158.623,108.803,-378.023,-1.6443,8.8235,-90.0002
C01373=2159.706,108.803,-378.052,0.2005,5.1337,-90.0002
C01374=2164.528,108.803,-377.988,-3.9247,4.0794,-90.0002
C01375=2165.061,108.803,-377.750,-1.7990,2.4751,-90.0002
C01376=2169.864,108.803,-377.381,-2.5038,3.5294,-90.0002
C01377=2170.425,108.803,-377.373,-0.0687,3.1111,-90.0002
C01378=2174.112,108.803,-377.090,-0.6932,8.3479,-90.0002
C01379=2174.902,108.803,-377.071,-2.4579,1.4954,-90.0002
C01380=2176.445,108.803,-376.837,-1.1516,6.5890,-90.0002
C01381=2178.587,108.803,-377.080,0.4927,5.5462,-90.0002
C01382=2179.426,108.803,-376.837,-1.4037,4.1596,-90.0002
C01383=2180.476,108.803,-376.384,-1.5469,8.3422,-90.0002
C01384=2181.164,108.803,-377.498,-1.1058,12.8399,-90.0002
C01385=2185.019,108.803,-375.142,-2.3147,16.4897,-90.0002
C01386=2185.530,108.803,-375.837,-0.0572,11.7685,-90.0002
C01387=2188.541,108.803,-375.235,-1.0886,-13.6363,-90.0002
C01388=2185.502,58.803,-375.622,-0.0515,2.0282,-90.0002
C01389=2184.587,58.803,-375.704,-1.1573,9.5110,-90.0002
C01390=2181.334,58.803,-375.888,-0.1203,9.2246,-90.0002
C01391=2180.186,58.803,-376.104,-1.3464,10.6169,-90.0002
C01392=2177.745,58.803,-376.686,1.9194,5.8728,-90.0002
C01393=2175.909,58.803,-376.663,-2.0855,0.2807,-90.0002
C01394=2174.454,58.803,-377.270,-1.8964,10.5309,-90.0002
C01395=2172.787,58.803,-376.982,0.5099,2.3147,-90.0002
C01396=2170.187,58.803,-377.417,3.0882,5.9301,-90.0002
C01397=2168.929,58.803,-377.238,0.8078,1.7818,-90.0002
C01398=2165.565,58.803,-377.616,1.5813,7.7922,-90.0002
C01399=2164.422,58.803,-377.925,0.4010,2.0569,-90.0002
C01400=2160.181,58.803,-377.880,-3.4721,0.5672,-90.0002
C01401=2159.040,58.803,-378.155,1.8105,3.7872,-90.0002
C01402=2155.756,58.803,-378.165,0.6187,5.9931,-90.0002
C01403=2154.515,58.803,-378.187,1.1172,-3.2257,-90.0002
C01404=2150.984,58.803,-378.776,-0.4526,7.3338,-90.0002
C01405=2149.951,58.803,-378.829,2.5611,2.4579,-90.0002
C01406=2145.683,58.803,-379.110,1.7933,0.4698,-90.0002
C01407=2143.964,58.803,-379.252,0.2578,2.0454,-90.0002
C01408=2140.681,58.803,-379.571,-0.4010,3.6382,-90.0002
C01409=2139.364,58.803,-379.434,-2.2574,2.5668,-90.0002
C01410=2135.250,58.803,-379.701,0.1661,5.9816,-90.0002
C01411=2134.565,58.803,-379.901,2.3433,2.2746,-90.0002
C01412=2130.555,58.803,-379.773,0.9740,1.0943,-90.0002
C01413=2128.778,58.803,-380.055,-1.3464,5.0993,-90.0002
C01414=2125.039,58.803,-379.997,-2.0053,1.4438,-90.0002
C01415=2123.450,58.803,-380.182,-2.3548,4.9675,-90.0002
C01416=2120.144,58.803,-380.051,1.0657,4.9675,-90.0002
C01417=2119.439,58.803,-380.544,-3.0022,6.8411,-90.0002
C01418=2115.315,58.803,-380.917,-1.4667,2.7559,-90.0002
C01419=2114.666,58.803,-380.805,-1.2204,4.4175,-90.0002
C01420=2110.782,58.803,-381.136,0.0515,-0.1489,-90.0002
C01421=2109.540,58.803,-380.902,1.2261,4.7326,-90.0002
C01422=2105.405,58.803,-381.373,-0.9740,-0.5156,-90.0002
C01423=2104.154,58.803,-381.173,-0.0802,3.3861,-90.0002
C01424=2100.313,58.803,-381.393,1.4438,-2.9392,-90.0002
C01425=2099.416,58.803,-381.361,3.1971,2.1886,-90.0002
C01426=2095.705,58.803,-381.541,-0.8651,2.2975,-90.0002
C01427=2094.399,58.803,-381.243,-1.9022,10.2444,-90.0002
C01428=2090.482,58.803,-381.699,0.5213,0.5385,-90.0002
C01429=2089.894,58.803,-381.726,-0.3437,7.0932,-90.0002
C01430=2088.622,58.803,-381.671,-4.8071,3.3116,-90.0002
C01431=2085.713,58.803,-381.989,2.5095,1.5813,-90.0002
C01432=2084.932,58.803,-382.119,2.4408,-3.5294,-90.0002
C01433=2083.804,58.803,-382.023,-3.0366,7.2937,-90.0002
C01434=2080.895,58.803,-382.327,-6.8640,7.6031,-90.0002
C01435=2079.430,58.803,-382.144,1.5412,0.1375,-90.0002
C01436=2076.700,58.803,-381.799,-1.1401,-1.6959,-90.0002
C01437=2075.381,58.803,-381.594,2.0741,2.6413,-90.0002
C01438=2074.734,58.803,-381.984,-0.4068,10.2043,-90.0002
C01439=2073.666,58.803,-381.686,1.0771,-1.7475,-90.0002
C01440=2070.998,58.803,-382.174,-2.3319,5.5806,-90.0002
C01441=2069.894,58.803,-382.356,0.0229,2.4121,-90.0002
C01442=2066.142,58.803,-381.817,2.8418,-7.8380,-90.0002
C01443=2065.130,58.803,-382.222,0.0000,4.9732,-90.0002
C01444=2064.109,58.803,-382.313,0.1317,0.0458,-90.0002
C01445=2059.976,58.803,-382.791,0.0171,2.4637,-90.0002
C01446=2059.344,58.803,-382.491,-1.6214,4.0049,-90.0002
C01447=2055.137,58.803,-382.767,0.2463,0.9281,-90.0002
C01448=2054.262,58.803,-382.732,-1.3980,9.6085,-90.0002
C01449=2050.756,58.803,-382.822,-1.2204,1.7990,-90.0002
C01450=2049.656,58.803,-382.466,-2.2689,4.7555,-90.0002
C01451=2045.238,58.803,-383.017,0.3495,2.3720,-90.0002
C01452=2044.711,58.803,-382.562,3.3346,0.1776,-90.0002
C01453=2040.460,58.803,-382.439,-3.6039,-0.0057,-90.0002
C01454=2039.362,58.803,-382.724,-3.8044,5.2425,-90.0002
C01455=2035.985,58.803,-382.893,0.5271,2.5382,-90.0002
C01456=2034.820,58.803,-382.546,1.3464,3.8101,-90.0002
C01457=2030.644,58.803,-382.672,0.8594,-1.0084,-90.0002
C01458=2030.169,58.803,-383.193,1.6214,1.1344,-90.0002
C01459=2025.187,58.803,-382.877,-0.0974,-1.7876,-90.0002
C01460=2024.574,58.803,-383.229,-0.0744,4.0049,-90.0002
C01461=2020.476,58.803,-383.039,-7.4312,2.6929,-90.0002
C01462=2019.466,58.803,-382.959,2.8074,-3.9304,-90.0002
C01463=2015.631,58.803,-382.903,-2.2861,1.4323,-90.0002
C01464=2015.048,58.803,-382.657,-0.3151,-0.9568,-90.0002
C01465=2010.573,58.803,-383.196,0.4354,-0.4812,-90.0002
C01466=2010.196,58.803,-383.078,1.5756,2.4293,-90.0002
C01467=2005.701,58.803,-383.121,-0.0229,-0.4182,-90.0002
C01468=2004.681,58.803,-382.914,1.6501,-0.4640,-90.0002
C01469=2000.403,58.803,-383.270,2.0168,0.6760,-90.0002
C01470=1999.773,58.803,-382.763,1.3636,-2.3147,-90.0002
C01471=1995.965,58.803,-383.525,1.7933,1.2662,-90.0002
C01472=1994.614,58.803,-383.090,-2.3262,3.8731,-90.0002
C01473=1990.010,58.803,-383.727,2.3491,1.1860,-90.0002
C01474=1989.339,58.803,-382.844,-7.9068,2.3835,-90.0002
C01475=1985.330,58.803,-383.000,-1.5412,4.2226,-90.0002
C01476=1984.855,58.803,-383.668,0.2750,-0.0859,-90.0002
C01477=1980.565,58.803,-383.301,1.7131,0.3093,-90.0002
C01478=1979.406,58.803,-383.427,-3.6210,-0.9167,-90.0002
C01479=1975.633,58.803,-383.409,0.7333,3.4262,-90.0002
C01480=1974.632,58.803,-383.625,-3.4721,-1.0084,-90.0002
C01481=1970.094,58.803,-383.404,-0.2979,3.3518,-90.0002
C01482=1969.228,58.803,-383.285,0.8078,-1.8048,-90.0002
C01483=1965.431,58.803,-383.353,0.9854,0.6818,-90.0002
C01484=1964.322,58.803,-383.483,0.4182,-0.8594,-90.0002
C01485=1960.406,58.803,-383.682,-0.3437,5.8155,-90.0002
C01486=1959.568,58.803,-383.464,0.5443,1.6386,-90.0002
C01487=1955.232,58.803,-383.720,-1.7074,0.1661,-90.0002
C01488=1954.550,58.803,-384.072,0.2291,0.1661,-90.0002
C01489=1950.253,58.803,-383.661,-2.1428,3.9591,-90.0002
C01490=1949.237,58.803,-383.741,-0.9912,-0.7964,-90.0002
C01491=1945.042,58.803,-383.696,0.8938,2.8304,-90.0002
C01492=1944.229,58.803,-383.864,-0.1031,-1.5126,-90.0002
C01493=1940.243,58.803,-383.674,0.8537,0.2234,-90.0002
C01494=1939.598,58.803,-383.521,-2.8991,0.7219,-90.0002
C01495=1934.733,58.803,-383.900,1.1802,0.7104,-90.0002
C01496=1934.150,58.803,-383.736,2.5439,-1.2204,-90.0002
C01497=1929.731,58.803,-383.984,1.6501,-1.0886,-90.0002
C01498=1928.887,58.803,-383.919,1.6157,2.3204,-90.0002
C01499=1925.319,58.803,-384.022,1.2948,0.9740,-90.0002
C01500=1924.421,58.803,-383.615,-0.2692,0.3208,-90.0002
C01501=1920.347,58.803,-383.889,-2.5095,-2.2173,-90.0002
C01502=1918.947,58.803,-383.934,-1.3292,2.9793,-90.0002
C01503=1915.472,58.803,-383.526,2.9851,-2.6298,-90.0002
C01504=1914.276,58.803,-383.502,1.8449,4.4862,-90.0002
C01505=1910.641,58.803,-383.604,-0.3953,-1.4667,-90.0002
C01506=1908.610,58.803,-383.777,0.7906,2.9163,-90.0002
C01507=1904.933,58.803,-383.473,2.3262,0.3781,-90.0002
C01508=1903.988,58.803,-383.867,1.2605,-4.3831,-90.0002
C01509=1899.603,58.803,-383.901,0.2119,-1.2032,-90.0002
C01510=1899.065,58.803,-383.767,-3.4663,-0.6646,-90.0002
C01511=1894.408,58.803,-383.572,-0.9969,0.1546,-90.0002
C01512=1893.986,58.803,-383.686,1.3120,-1.4266,-90.0002
C01513=1890.113,58.803,-383.601,-2.5324,-3.6554,-90.0002
C01514=1885.581,58.803,-383.341,-0.5958,-1.2948,-90.0002
C01515=1885.101,58.803,-383.330,-3.2830,0.3609,-90.0002
C01516=1881.620,58.803,-382.819,1.8678,-2.0741,-90.0002
C01517=1879.575,58.803,-383.315,-2.7387,-4.8873,-90.0002
C01518=1875.961,58.803,-383.349,0.2406,0.0630,-90.0002
C01519=1875.053,58.803,-383.258,-1.1058,1.4381,-90.0002
C01520=1871.217,58.803,-383.091,0.4870,0.8479,-90.0002
C01521=1870.023,58.803,-382.821,-4.8529,-4.5206,-90.0002
C01522=1865.779,58.803,-382.711,-2.0282,-3.3059,-90.0002
C01523=1864.214,58.803,-382.880,0.3265,-1.7704,-90.0002
C01524=1860.166,58.803,-382.494,-1.9308,-0.3036,-90.0002
C01525=1859.143,58.803,-382.129,1.6558,-4.6008,-90.0002
C01526=1856.059,58.803,-382.618,-0.7906,-1.1917,-90.0002
C01527=1854.337,58.803,-381.870,2.0053,1.0542,-90.0002
C01528=1852.620,58.803,-382.149,-0.1317,-5.4144,-90.0002
C01529=1850.548,58.803,-382.288,-0.3724,-3.1111,-90.0002
C01530=1849.250,58.803,-382.128,3.5523,-3.7929,-90.0002
C01531=1847.930,58.803,-381.849,2.2631,-4.4805,-90.0002
C01532=1845.672,58.803,-381.812,-2.2230,-3.8388,-90.0002
C01533=1844.518,58.803,-381.759,-1.0542,-5.7868,-90.0002
C01534=1842.170,58.803,-381.737,0.1375,-1.7303,-90.0002
C01535=1839.610,58.803,-381.495,-0.3838,-3.0366,-90.0002
C01536=1835.873,58.803,-381.287,-0.2005,-4.1482,-90.0002
C01537=1834.250,58.803,-381.223,-0.1432,-4.7956,-90.0002
C01538=1830.424,58.803,-381.145,1.5412,-4.7154,-90.0002
C01539=1829.330,58.803,-380.908,-0.1203,-3.2429,-90.0002
C01540=1825.463,58.803,-380.787,2.7272,-5.3456,-90.0002
C01541=1824.811,58.803,-380.790,0.4469,-3.7815,-90.0002
C01542=1820.697,58.803,-380.122,-4.4117,-2.3090,-90.0002
C01543=1820.073,58.803,-380.341,-1.3464,-3.7872,-90.0002
C01544=1815.208,58.803,-379.935,1.1287,-0.7219,-90.0002
C01545=1813.968,58.803,-379.830,-3.1226,-1.7818,-90.0002
C01546=1810.175,58.803,-379.725,-3.4320,-5.0420,-90.0002
C01547=1809.588,58.803,-379.670,0.8479,-6.0389,-90.0002
C01548=1805.581,58.803,-379.087,-0.4583,-7.1562,-90.0002
C01549=1804.197,58.803,-379.105,4.4690,-6.9786,-90.0002
C01550=1800.624,58.803,-378.792,1.5469,-3.5523,-90.0002
C01551=1800.080,58.803,-378.764,-2.0912,-5.7983,-90.0002
C01552=1795.146,58.803,-377.697,1.4725,-12.3300,-90.0002
C01553=1798.894,8.803,-378.601,-3.4893,-5.5576,-90.0002
C01554=1799.874,8.803,-378.703,-0.9052,-2.7903,-90.0002
C01555=1803.731,8.803,-378.851,-0.5271,-8.5428,-90.0002
C01556=1804.996,8.803,-379.130,1.1172,-9.4194,-90.0002
C01557=1808.212,8.803,-379.516,0.4526,-4.9961,-90.0002
C01558=1810.246,8.803,-379.250,1.0026,-4.3659,-90.0002
C01559=1813.388,8.803,-379.809,-6.3025,0.7734,-90.0002
C01560=1814.666,8.803,-379.843,1.4037,-3.5065,-90.0002
C01561=1817.731,8.803,-379.844,1.5183,-4.3086,-90.0002
C01562=1819.765,8.803,-380.143,1.3693,-0.4354,-90.0002
C01563=1823.736,8.803,-380.365,0.6474,-3.4262,-90.0002
C01564=1825.030,8.803,-380.140,-0.2005,-2.8017,-90.0002
C01565=1829.030,8.803,-381.056,1.2948,-3.7242,-90.0002
C01566=1830.159,8.803,-380.847,0.9568,-3.3976,-90.0002
C01567=1833.665,8.803,-381.235,-1.3865,2.4923,-90.0002
C01568=1834.861,8.803,-381.245,2.8418,-0.7505,-90.0002
C01569=1838.641,8.803,-381.487,1.6673,-4.5378,-90.0002
C01570=1839.725,8.803,-381.101,-1.6558,-0.4583,-90.0002
C01571=1840.896,8.803,-381.998,-2.7043,-9.4996,-90.0002
C01572=1844.249,8.803,-381.278,-1.7074,-1.6443,-90.0002
C01573=1845.828,8.803,-381.090,-0.4469,-2.9564,-90.0002
C01574=1848.645,8.803,-381.508,1.6844,-4.7727,-90.0002
C01575=1849.939,8.803,-381.733,1.7589,2.0970,-90.0002
C01576=1851.853,8.803,-381.959,-0.0687,-1.3521,-90.0002
C01577=1854.092,8.803,-382.227,-0.2234,-2.0970,-90.0002
C01578=1855.033,8.803,-381.980,-1.2547,-1.2032,-90.0002
C01579=1858.951,8.803,-381.746,4.7269,-0.5614,-90.0002
C01580=1860.353,8.803,-382.463,-0.3036,-3.0939,-90.0002
C01581=1861.721,8.803,-382.169,2.0225,0.0458,-90.0002
C01582=1865.128,8.803,-382.819,3.4663,-3.5752,-90.0002
C01583=1866.119,8.803,-381.824,0.0000,2.4350,-90.0002
C01584=1869.238,8.803,-383.038,0.3093,-4.1596,-90.0002
C01585=1869.781,8.803,-382.206,3.2085,-1.4381,-90.0002
C01586=1874.067,8.803,-382.729,2.1371,2.9736,-90.0002
C01587=1874.982,8.803,-382.825,0.0687,-0.5443,-90.0002
C01588=1877.430,8.803,-382.695,1.4152,-1.9767,-90.0002
C01589=1880.280,8.803,-382.513,-0.8766,-1.6902,-90.0002
C01590=1881.633,8.803,-382.741,-2.6298,-3.5752,-90.0002
C01591=1884.822,8.803,-383.129,-0.3380,-0.9625,-90.0002
C01592=1886.160,8.803,-382.472,-1.5469,2.1428,-90.0002
C01593=1890.121,8.803,-383.547,1.5240,-0.6474,-90.0002
C01594=1891.232,8.803,-383.371,1.0026,-2.3204,-90.0002
C01595=1895.136,8.803,-383.093,-2.0741,0.7906,-90.0002
C01596=1896.427,8.803,-383.638,3.9705,-3.4778,-90.0002
C01597=1899.180,8.803,-383.160,0.0687,-1.2547,-90.0002
C01598=1900.888,8.803,-382.681,3.1340,-2.8705,-90.0002
C01599=1904.903,8.803,-383.065,1.2490,0.4755,-90.0002
C01600=1905.816,8.803,-382.772,2.9564,-0.0114,-90.0002
C01601=1909.631,8.803,-382.819,-2.6470,2.6126,-90.0002
C01602=1914.174,8.803,-382.556,5.8785,0.3724,-90.0002
C01603=1915.668,8.803,-383.397,4.3487,-1.5756,-90.0002
C01604=1918.191,8.803,-382.853,-0.9568,0.4125,-90.0002
C01605=1920.545,8.803,-383.109,1.5813,0.1890,-90.0002
C01606=1923.828,8.803,-383.561,-0.3265,2.0110,-90.0002
C01607=1925.621,8.803,-383.491,2.8189,0.6932,-90.0002
C01608=1928.924,8.803,-383.132,4.1539,2.4809,-90.0002
C01609=1930.221,8.803,-383.050,3.5867,-0.6760,-90.0002
C01610=1934.139,8.803,-382.735,1.9767,0.9912,-90.0002
C01611=1935.506,8.803,-382.861,4.4518,-4.9274,-90.0002
C01612=1938.911,8.803,-382.668,5.7123,3.2429,-90.0002
C01613=1939.988,8.803,-382.986,2.0798,-6.8583,-90.0002
C01614=1944.067,8.803,-382.539,0.5156,-1.0198,-90.0002
C01615=1945.073,8.803,-381.750,3.4721,-2.3949,-90.0002
C01616=1948.562,8.803,-383.489,5.8269,-3.8846,-90.0002
C01617=1949.549,8.803,-383.018,-0.7391,1.7990,-90.0002
C01618=1951.671,8.803,-381.909,2.8762,0.6073,-90.0002
C01619=1954.708,8.803,-382.811,-0.4640,1.0084,-90.0002
C01620=1956.281,8.803,-382.140,1.5068,-0.0171,-90.0002
C01621=1959.804,8.803,-382.649,-0.1432,3.5523,-90.0002
C01622=1960.634,8.803,-382.671,3.9190,3.0194,-90.0002
C01623=1964.757,8.803,-383.227,1.5527,0.8594,-90.0002
C01624=1965.783,8.803,-382.461,-0.2062,1.5641,-90.0002
C01625=1969.332,8.803,-382.489,-2.5152,-1.7532,-90.0002
C01626=1970.399,8.803,-382.187,4.4862,1.4954,-90.0002
C01627=1974.685,8.803,-382.745,2.1543,3.0366,-90.0002
C01628=1975.213,8.803,-382.463,2.7559,-0.0515,-90.0002
C01629=1979.096,8.803,-383.224,-0.5729,6.2165,-90.0002
C01630=1980.965,8.803,-382.278,5.2196,-0.8136,-90.0002
C01631=1983.944,8.803,-382.980,-3.4606,2.9048,-90.0002
C01632=1985.069,8.803,-383.157,2.1944,-5.3055,-90.0002
C01633=1988.765,8.803,-382.456,-0.2349,-2.0282,-90.0002
C01634=1989.888,8.803,-382.090,1.8563,1.4323,-90.0002
C01635=1990.341,8.803,-382.930,1.4094,4.9961,-90.0002
C01636=1993.928,8.803,-382.864,-0.7563,-2.8304,-90.0002
C01637=1995.346,8.803,-383.412,2.8074,4.2685,-90.0002
C01638=1999.376,8.803,-382.764,4.6352,4.5550,-90.0002
C01639=1999.957,8.803,-382.491,1.4782,1.3521,-90.0002
C01640=2001.129,8.803,-381.640,-6.1306,0.4870,-90.0002
C01641=2003.744,8.803,-383.015,-6.2910,4.0565,-90.0002
C01642=2005.057,8.803,-382.069,-0.6875,6.8812,-90.0002
C01643=2008.712,8.803,-382.085,4.8128,1.4037,-90.0002
C01644=2009.806,8.803,-382.878,-0.4812,5.0764,-90.0002
C01645=2012.925,8.803,-381.918,-1.8563,-0.9682,-90.0002
C01646=2015.064,8.803,-382.624,1.4381,-0.1890,-90.0002
C01647=2016.149,8.803,-382.482,-4.3201,4.4404,-90.0002
C01648=2018.113,8.803,-382.473,4.5664,2.9736,-90.0002
C01649=2019.538,8.803,-382.127,1.3407,2.3090,-90.0002
C01650=2020.615,8.803,-382.598,-0.1031,-2.8533,-90.0002
C01651=2023.397,8.803,-381.921,2.2689,6.8640,-90.0002
C01652=2025.430,8.803,-381.853,-0.4526,8.8235,-90.0002
C01653=2026.143,8.803,-382.299,-1.0943,-6.1707,-90.0002
C01654=2029.744,8.803,-381.628,3.5065,-0.0802,-90.0002
C01655=2030.943,8.803,-382.368,1.3292,-2.3204,-90.0002
C01656=2033.843,8.803,-381.831,-4.9159,1.0599,-90.0002
C01657=2035.120,8.803,-381.854,3.1913,1.6329,-90.0002
C01658=2036.216,8.803,-381.666,2.6642,1.2547,-90.0002
C01659=2039.656,8.803,-382.222,2.1142,1.0370,-90.0002
C01660=2040.336,8.803,-382.027,4.6237,3.9304,-90.0002
C01661=2044.682,8.803,-381.296,0.9740,0.7505,-90.0002
C01662=2045.132,8.803,-382.311,1.1573,2.5496,-90.0002
C01663=2046.168,8.803,-382.433,-0.9224,0.7161,-90.0002
C01664=2049.178,8.803,-382.426,0.9052,7.4312,-90.0002
C01665=2050.186,8.803,-381.789,1.6501,3.8789,-90.0002
C01666=2051.798,8.803,-381.716,0.4812,5.9587,-90.0002
C01667=2053.688,8.803,-382.030,1.7246,2.1371,-90.0002
C01668=2054.878,8.803,-381.594,1.3636,2.7845,-90.0002
C01669=2056.375,8.803,-381.770,0.9511,0.1375,-90.0002
C01670=2058.327,8.803,-381.651,2.6757,-5.8670,-90.0002
C01671=2059.785,8.803,-382.200,0.1546,-0.2692,-90.0002
C01672=2061.250,8.803,-381.756,3.2142,2.1142,-90.0002
C01673=2063.874,8.803,-382.207,-3.6440,1.5699,-90.0002
C01674=2065.184,8.803,-382.199,0.7219,-0.8250,-90.0002
C01675=2066.546,8.803,-382.027,1.5641,-0.0802,-90.0002
C01676=2069.277,8.803,-381.350,-1.2261,-1.4495,-90.0002
C01677=2070.702,8.803,-381.843,0.9797,4.1023,-90.0002
C01678=2071.873,8.803,-381.587,-0.0286,7.5229,-90.0002
C01679=2074.360,8.803,-381.986,1.3349,2.5611,-90.0002
C01680=2075.422,8.803,-381.676,2.0110,7.7864,-90.0002
C01681=2078.932,8.803,-381.534,3.1455,-1.0026,-90.0002
C01682=2079.949,8.803,-381.507,2.6356,-5.3055,-90.0002
C01683=2084.420,8.803,-381.675,4.3544,-3.8445,-90.0002
C01684=2085.146,8.803,-381.581,1.9136,2.9851,-90.0002
C01685=2087.746,8.803,-381.366,0.4984,-0.2291,-90.0002
C01686=2089.249,8.803,-380.882,1.7704,2.8590,-90.0002
C01687=2090.194,8.803,-382.156,2.7731,2.3720,-90.0002
C01688=2094.465,8.803,-380.936,-2.4236,2.9450,-90.0002
C01689=2096.081,8.803,-381.151,2.2574,-1.3808,-90.0002
C01690=2099.895,8.803,-381.059,1.0427,-0.9511,-90.0002
C01691=2101.198,8.803,-380.864,2.3720,9.5168,-90.0002
C01692=2105.068,8.803,-381.276,4.0622,4.3602,-90.0002
C01693=2106.438,8.803,-380.837,-0.6130,1.6558,-90.0002
C01694=2109.528,8.803,-380.861,0.7047,1.4495,-90.0002
C01695=2110.846,8.803,-380.588,0.1088,7.0416,-90.0002
C01696=2114.640,8.803,-380.177,-0.2177,2.5038,-90.0002
C01697=2115.458,8.803,-380.384,-0.0171,6.2051,-90.0002
C01698=2119.588,8.803,-379.801,1.0886,1.2204,-90.0002
C01699=2121.498,8.803,-379.873,2.8476,2.3548,-90.0002
C01700=2124.614,8.803,-379.701,-0.2979,0.1031,-90.0002
C01701=2126.311,8.803,-379.634,1.3636,6.6864,-90.0002
C01702=2130.106,8.803,-379.760,0.8021,2.3090,-90.0002
C01703=2133.256,8.803,-379.607,-1.1401,3.0825,-90.0002
C01704=2135.454,8.803,-379.716,1.4667,5.6035,-90.0002
C01705=2138.900,8.803,-379.399,-0.9740,1.8563,-90.0002
C01706=2140.496,8.803,-379.454,1.8277,1.9022,-90.0002
C01707=2143.219,8.803,-379.253,-1.1344,5.6149,-90.0002
C01708=2144.888,8.803,-378.834,-3.1971,6.6520,-90.0002
C01709=2148.266,8.803,-379.009,2.2746,2.1027,-90.0002
C01710=2149.837,8.803,-378.563,0.7047,0.7792,-90.0002
C01711=2154.077,8.803,-378.213,1.5584,4.5893,-90.0002
C01712=2155.082,8.803,-378.577,-0.0630,6.5431,-90.0002
C01713=2158.906,8.803,-377.860,-1.8735,3.3747,-90.0002
C01714=2160.225,8.803,-378.014,-1.9480,3.0939,-90.0002
C01715=2163.890,8.803,-377.623,0.6474,5.6149,-90.0002
C01716=2164.880,8.803,-377.783,1.6214,3.8445,-90.0002
C01717=2169.386,8.803,-377.358,-4.2628,2.0741,-90.0002
C01718=2170.175,8.803,-377.246,-1.4896,0.3838,-90.0002
C01719=2171.774,8.803,-376.772,-2.7960,6.1936,-90.0002
C01720=2174.349,8.803,-377.086,0.0171,4.6581,-90.0002
C01721=2175.360,8.803,-377.013,1.9136,6.6749,-90.0002
C01722=2177.008,8.803,-377.163,-7.4541,1.8964,-90.0002
C01723=2180.561,8.803,-376.316,-0.1718,10.0439,-90.0002
C01724=2181.078,8.803,-376.110,-2.2861,5.0764,-90.0002
C01725=2184.526,8.803,-375.725,-4.3143,8.3078,-90.0002
C01726=2185.880,-41.196,-375.195,-1.1172,8.6000,-90.0002
C01727=2184.495,-41.196,-375.702,-1.5240,7.4484,-90.0002
C01728=2181.254,-41.196,-376.002,-1.1802,5.1337,-90.0002
C01729=2179.901,-41.196,-376.252,-4.8816,5.9530,-90.0002
C01730=2177.291,-41.196,-376.736,-0.5042,5.4316,-90.0002
C01731=2174.987,-41.196,-377.102,-0.2635,6.4056,-90.0002
C01732=2173.467,-41.196,-377.244,-0.0171,6.3655,-90.0002
C01733=2170.873,-41.196,-376.921,-0.3495,3.7127,-90.0002
